LIN {X 0,Y 218.448,Z 342.659,A -85,B 0,C 180,E1 -22368.616,E2 -22368.616} C_VEL
LIN {X 0,Y 217.476,Z 348.635,A -85,B 0,C 180,E1 -22368.653,E2 -22368.653} C_VEL
LIN {X 0,Y 215.786,Z 367.504,A -85,B 0,C 180,E1 -22369.355,E2 -22369.355} C_VEL
LIN {X 0,Y 213.676,Z 380.389,A -85,B 0,C 180,E1 -22370.107,E2 -22370.107} C_VEL
LIN {X 0,Y 210.515,Z 393.733,A -85,B 0,C 180,E1 -22371.248,E2 -22371.248} C_VEL
LIN {X 0,Y 207.06,Z 405.5,A -85,B 0,C 180,E1 -22372.649,E2 -22372.649} C_VEL
LIN {X 0,Y 203.22,Z 416.165,A -85,B 0,C 180,E1 -22374.298,E2 -22374.298} C_VEL
LIN {X 0,Y 199.229,Z 425.901,A -85,B 0,C 180,E1 -22376.249,E2 -22376.249} C_VEL
LIN {X 0,Y 195.179,Z 434.841,A -85,B 0,C 180,E1 -22378.527,E2 -22378.527} C_VEL
LIN {X 0,Y 190.718,Z 443.631,A -85,B 0,C 180,E1 -22381.377,E2 -22381.377} C_VEL
LIN {X 0,Y 186.992,Z 450.647,A -85,B 0,C 180,E1 -22384.353,E2 -22384.353} C_VEL
LIN {X 0,Y 183.667,Z 456.423,A -85,B 0,C 180,E1 -22387.503,E2 -22387.503} C_VEL
LIN {X 0,Y 180.963,Z 460.965,A -85,B 0,C 180,E1 -22390.725,E2 -22390.725} C_VEL
LIN {X 0,Y 178.739,Z 464.46,A -85,B 0,C 180,E1 -22394.024,E2 -22394.024} C_VEL
LIN {X 0,Y 176.979,Z 467.604,A -85,B 0,C 180,E1 -22398.548,E2 -22398.548} C_VEL
LIN {X 0,Y 176.111,Z 469.188,A -85,B 0,C 180,E1 -22403.124,E2 -22403.124} C_VEL
LIN {X 0,Y 175.999,Z 469.294,A -85,B 0,C 180,E1 -22406.825,E2 -22406.825} C_VEL
LIN {X 0,Y 176.229,Z 468.533,A -85,B 0,C 180,E1 -22410,E2 -22410} C_VEL
LIN {X 0,Y 176.089,Z 466.648,A -85,B 0,C 180,E1 -22413.663,E2 -22413.663} C_VEL
LIN {X 0,Y 176.336,Z 462.93,A -85,B 0,C 180,E1 -22418.019,E2 -22418.019} C_VEL
LIN {X 0,Y 176.923,Z 458.748,A -85,B 0,C 180,E1 -22421.456,E2 -22421.456} C_VEL
LIN {X 0,Y 178.216,Z 452.316,A -85,B 0,C 180,E1 -22425.437,E2 -22425.437} C_VEL
LIN {X 0,Y 180.018,Z 445.292,A -85,B 0,C 180,E1 -22428.789,E2 -22428.789} C_VEL
LIN {X 0,Y 181.778,Z 438.618,A -85,B 0,C 180,E1 -22431.344,E2 -22431.344} C_VEL
LIN {X 0,Y 184.193,Z 429.348,A -85,B 0,C 180,E1 -22434.215,E2 -22434.215} C_VEL
LIN {X 0,Y 186.584,Z 419.767,A -85,B 0,C 180,E1 -22436.569,E2 -22436.569} C_VEL
LIN {X 0,Y 188.379,Z 412.204,A -85,B 0,C 180,E1 -22438.099,E2 -22438.099} C_VEL
LIN {X 0,Y 190.939,Z 399.705,A -85,B 0,C 180,E1 -22440.099,E2 -22440.099} C_VEL
LIN {X 0,Y 193.124,Z 387.562,A -85,B 0,C 180,E1 -22441.541,E2 -22441.541} C_VEL
LIN {X 0,Y 194.875,Z 374.064,A -85,B 0,C 180,E1 -22442.672,E2 -22442.672} C_VEL
LIN {X 0,Y 196.016,Z 361.06,A -85,B 0,C 180,E1 -22443.361,E2 -22443.361} C_VEL
LIN {X 0,Y 198.16,Z 316.515,A -85,B 0,C 180,E1 -22445.049,E2 -22445.049} C_VEL
LIN {X 0,Y 195.778,Z 296.397,A -85,B 0,C 180,E1 -22446.33,E2 -22446.33} C_VEL
LIN {X 0,Y 188.073,Z 275.885,A -85,B 0,C 180,E1 -22448.617,E2 -22448.617} C_VEL
LIN {X 0,Y 181.122,Z 260.53,A -85,B 0,C 180,E1 -22450.71,E2 -22450.71} C_VEL
LIN {X 0,Y 179.58,Z 257.045,A -85,B 0,C 180,E1 -22451.221,E2 -22451.221} C_VEL
LIN {X 0,Y 178.411,Z 252.269,A -85,B 0,C 180,E1 -22454.021,E2 -22454.021} C_VEL
LIN {X 0,Y 178.409,Z 252.262,A -85,B 0,C 180,E1 -22458.456,E2 -22458.456} C_VEL
LIN {X 0,Y 178.434,Z 252.257,A -85,B 0,C 180,E1 -22463.773,E2 -22463.773} C_VEL
LIN {X 0,Y 178.497,Z 252.253,A -85,B 0,C 180,E1 -22466.536,E2 -22466.536} C_VEL
LIN {X 0,Y 178.432,Z 252.258,A -85,B 0,C 180,E1 -22471.781,E2 -22471.781} C_VEL
LIN {X 0,Y 178.473,Z 252.253,A -85,B 0,C 180,E1 -22476.797,E2 -22476.797} C_VEL
LIN {X 0,Y 178.613,Z 252.201,A -85,B 0,C 180,E1 -22481.64,E2 -22481.64} C_VEL
LIN {X 0,Y 178.64,Z 252.227,A -85,B 0,C 180,E1 -22486.334,E2 -22486.334} C_VEL
LIN {X 0,Y 178.902,Z 252.196,A -85,B 0,C 180,E1 -22490.947,E2 -22490.947} C_VEL
LIN {X 0,Y 179.098,Z 252.128,A -85,B 0,C 180,E1 -22497.738,E2 -22497.738} C_VEL
LIN {X 0,Y 179.333,Z 252.122,A -85,B 0,C 180,E1 -22499.987,E2 -22499.987} C_VEL
LIN {X 0,Y 178.824,Z 252.209,A -85,B 0,C 180,E1 -22504.495,E2 -22504.495} C_VEL
LIN {X 0,Y 178.893,Z 252.189,A -85,B 0,C 180,E1 -22509.028,E2 -22509.028} C_VEL
LIN {X 0,Y 178.636,Z 252.234,A -85,B 0,C 180,E1 -22513.64,E2 -22513.64} C_VEL
LIN {X 0,Y 178.603,Z 252.223,A -85,B 0,C 180,E1 -22519.2,E2 -22519.2} C_VEL
LIN {X 0,Y 178.497,Z 252.245,A -85,B 0,C 180,E1 -22525.101,E2 -22525.101} C_VEL
LIN {X 0,Y 178.437,Z 252.208,A -85,B 0,C 180,E1 -22530.782,E2 -22530.782} C_VEL
LIN {X 0,Y 178.453,Z 252.224,A -85,B 0,C 180,E1 -22534.206,E2 -22534.206} C_VEL
LIN {X 0,Y 178.356,Z 252.267,A -85,B 0,C 180,E1 -22539.065,E2 -22539.065} C_VEL
LIN {X 0,Y 178.361,Z 252.261,A -85,B 0,C 180,E1 -22542.036,E2 -22542.036} C_VEL
LIN {X 0,Y 178.357,Z 252.263,A -85,B 0,C 180,E1 -22545.154,E2 -22545.154} C_VEL
LIN {X 0,Y 178.365,Z 252.265,A -85,B 0,C 180,E1 -22548.45,E2 -22548.45} C_VEL
LIN {X 0,Y 178.381,Z 252.266,A -85,B 0,C 180,E1 -22553.774,E2 -22553.774} C_VEL
LIN {X 0,Y 178.443,Z 252.252,A -85,B 0,C 180,E1 -22556.538,E2 -22556.538} C_VEL
LIN {X 0,Y 178.479,Z 252.256,A -85,B 0,C 180,E1 -22560,E2 -22560} C_VEL
LIN {X 0,Y 178.5,Z 252.256,A -85,B 0,C 180,E1 -22564.863,E2 -22564.863} C_VEL
LIN {X 0,Y 178.608,Z 252.243,A -85,B 0,C 180,E1 -22570.75,E2 -22570.75} C_VEL
LIN {X 0,Y 178.626,Z 252.239,A -85,B 0,C 180,E1 -22574.014,E2 -22574.014} C_VEL
LIN {X 0,Y 178.81,Z 252.209,A -85,B 0,C 180,E1 -22579.213,E2 -22579.213} C_VEL
LIN {X 0,Y 178.907,Z 252.197,A -85,B 0,C 180,E1 -22582.026,E2 -22582.026} C_VEL
LIN {X 0,Y 179.914,Z 255.085,A -85,B 0,C 180,E1 -22582.417,E2 -22582.417} C_VEL
LIN {X 0,Y 181.316,Z 257.484,A -85,B 0,C 180,E1 -22582.826,E2 -22582.826} C_VEL
LIN {X 0,Y 189.994,Z 273.152,A -85,B 0,C 180,E1 -22585.256,E2 -22585.256} C_VEL
LIN {X 0,Y 194.262,Z 282.713,A -85,B 0,C 180,E1 -22586.448,E2 -22586.448} C_VEL
LIN {X 0,Y 199.123,Z 295.475,A -85,B 0,C 180,E1 -22587.811,E2 -22587.811} C_VEL
LIN {X 0,Y 195.994,Z 353.238,A -85,B 0,C 180,E1 -22590,E2 -22590} C_VEL
LIN {X 0,Y 194.697,Z 366.02,A -85,B 0,C 180,E1 -22590.84,E2 -22590.84} C_VEL
LIN {X 0,Y 193.136,Z 378.634,A -85,B 0,C 180,E1 -22592.085,E2 -22592.085} C_VEL
LIN {X 0,Y 191.05,Z 390.66,A -85,B 0,C 180,E1 -22593.691,E2 -22593.691} C_VEL
LIN {X 0,Y 188.528,Z 402.811,A -85,B 0,C 180,E1 -22595.83,E2 -22595.83} C_VEL
LIN {X 0,Y 186.128,Z 413.03,A -85,B 0,C 180,E1 -22598.14,E2 -22598.14} C_VEL
LIN {X 0,Y 183.418,Z 423.131,A -85,B 0,C 180,E1 -22601.045,E2 -22601.045} C_VEL
LIN {X 0,Y 181.186,Z 431.752,A -85,B 0,C 180,E1 -22604.201,E2 -22604.201} C_VEL
LIN {X 0,Y 179.205,Z 439.195,A -85,B 0,C 180,E1 -22607.694,E2 -22607.694} C_VEL
LIN {X 0,Y 177.904,Z 444.467,A -85,B 0,C 180,E1 -22610.826,E2 -22610.826} C_VEL
LIN {X 0,Y 176.83,Z 449.719,A -85,B 0,C 180,E1 -22614.916,E2 -22614.916} C_VEL
LIN {X 0,Y 176.035,Z 453.133,A -85,B 0,C 180,E1 -22618.625,E2 -22618.625} C_VEL
LIN {X 0,Y 175.672,Z 455.615,A -85,B 0,C 180,E1 -22622.875,E2 -22622.875} C_VEL
LIN {X 0,Y 175.993,Z 456.678,A -85,B 0,C 180,E1 -22627.023,E2 -22627.023} C_VEL
LIN {X 0,Y 176.857,Z 456.49,A -85,B 0,C 180,E1 -22630.996,E2 -22630.996} C_VEL
LIN {X 0,Y 178.438,Z 455.004,A -85,B 0,C 180,E1 -22635.148,E2 -22635.148} C_VEL
LIN {X 0,Y 180.843,Z 451.875,A -85,B 0,C 180,E1 -22639.502,E2 -22639.502} C_VEL
LIN {X 0,Y 183.816,Z 447.528,A -85,B 0,C 180,E1 -22643.407,E2 -22643.407} C_VEL
LIN {X 0,Y 187.038,Z 442.414,A -85,B 0,C 180,E1 -22646.722,E2 -22646.722} C_VEL
LIN {X 0,Y 190.908,Z 435.903,A -85,B 0,C 180,E1 -22649.891,E2 -22649.891} C_VEL
LIN {X 0,Y 194.765,Z 428.674,A -85,B 0,C 180,E1 -22652.617,E2 -22652.617} C_VEL
LIN {X 0,Y 199.095,Z 419.632,A -85,B 0,C 180,E1 -22655.279,E2 -22655.279} C_VEL
LIN {X 0,Y 203.103,Z 410.186,A -85,B 0,C 180,E1 -22657.463,E2 -22657.463} C_VEL
LIN {X 0,Y 206.676,Z 400.411,A -85,B 0,C 180,E1 -22659.246,E2 -22659.246} C_VEL
LIN {X 0,Y 210.237,Z 388.81,A -85,B 0,C 180,E1 -22660.877,E2 -22660.877} C_VEL
LIN {X 0,Y 213.117,Z 377.076,A -85,B 0,C 180,E1 -22662.134,E2 -22662.134} C_VEL
LIN {X 0,Y 215.495,Z 364.012,A -85,B 0,C 180,E1 -22663.149,E2 -22663.149} C_VEL
LIN {X 0,Y 217.106,Z 350.758,A -85,B 0,C 180,E1 -22663.799,E2 -22663.799} C_VEL
LIN {X 0,Y 220.108,Z 311.417,A -85,B 0,C 180,E1 -22665.133,E2 -22665.133} C_VEL
LIN {X 0,Y 216.218,Z 302.782,A -85,B 0,C 180,E1 -22667.007,E2 -22667.007} C_VEL
LIN {X 0,Y 213.125,Z 297.063,A -85,B 0,C 180,E1 -22668.556,E2 -22668.556} C_VEL
LIN {X 0,Y 209.272,Z 290.775,A -85,B 0,C 180,E1 -22670.62,E2 -22670.62} C_VEL
LIN {X 0,Y 204.339,Z 283.304,A -85,B 0,C 180,E1 -22673.596,E2 -22673.596} C_VEL
LIN {X 0,Y 201.792,Z 279.641,A -85,B 0,C 180,E1 -22675.355,E2 -22675.355} C_VEL
LIN {X 0,Y 199.009,Z 276.05,A -85,B 0,C 180,E1 -22677.458,E2 -22677.458} C_VEL
LIN {X 0,Y 198.122,Z 274.662,A -85,B 0,C 180,E1 -22678.233,E2 -22678.233} C_VEL
LIN {X 0,Y 195.806,Z 271.796,A -85,B 0,C 180,E1 -22680.344,E2 -22680.344} C_VEL
LIN {X 0,Y 194.667,Z 269.788,A -85,B 0,C 180,E1 -22681.573,E2 -22681.573} C_VEL
LIN {X 0,Y 191.537,Z 267.402,A -85,B 0,C 180,E1 -22685.275,E2 -22685.275} C_VEL
LIN {X 0,Y 190.259,Z 264.56,A -85,B 0,C 180,E1 -22687.635,E2 -22687.635} C_VEL
LIN {X 0,Y 188.459,Z 263.748,A -85,B 0,C 180,E1 -22691.847,E2 -22691.847} C_VEL
LIN {X 0,Y 187.853,Z 263.472,A -85,B 0,C 180,E1 -22697.427,E2 -22697.427} C_VEL
LIN {X 0,Y 189.234,Z 264.37,A -85,B 0,C 180,E1 -22702.926,E2 -22702.926} C_VEL
LIN {X 0,Y 190.557,Z 266.295,A -85,B 0,C 180,E1 -22705.656,E2 -22705.656} C_VEL
LIN {X 0,Y 192.69,Z 269.516,A -85,B 0,C 180,E1 -22708.916,E2 -22708.916} C_VEL
LIN {X 0,Y 195.62,Z 273.297,A -85,B 0,C 180,E1 -22712.167,E2 -22712.167} C_VEL
LIN {X 0,Y 199.882,Z 279.881,A -85,B 0,C 180,E1 -22715.981,E2 -22715.981} C_VEL
LIN {X 0,Y 203.656,Z 286.092,A -85,B 0,C 180,E1 -22718.753,E2 -22718.753} C_VEL
LIN {X 0,Y 206.674,Z 291.312,A -85,B 0,C 180,E1 -22720.699,E2 -22720.699} C_VEL
LIN {X 0,Y 210.875,Z 299.125,A -85,B 0,C 180,E1 -22723.158,E2 -22723.158} C_VEL
LIN {X 0,Y 215.414,Z 308.937,A -85,B 0,C 180,E1 -22725.57,E2 -22725.57} C_VEL
LIN {X 0,Y 219.144,Z 318.713,A -85,B 0,C 180,E1 -22727.455,E2 -22727.455} C_VEL
LIN {X 0,Y 219.436,Z 321.912,A -85,B 0,C 180,E1 -22727.735,E2 -22727.735} C_VEL
LIN {X 0,Y 217.476,Z 348.635,A -85,B 0,C 180,E1 -22728.653,E2 -22728.653} C_VEL
LIN {X 0,Y 216.967,Z 352.543,A -85,B 0,C 180,E1 -22728.712,E2 -22728.712} C_VEL
LIN {X 0,Y 214.974,Z 360.206,A -85,B 0,C 180,E1 -22728.535,E2 -22728.535} C_VEL
LIN {X 0,Y 211.006,Z 371.945,A -85,B 0,C 180,E1 -22728.28,E2 -22728.28} C_VEL
LIN {X 0,Y 209.635,Z 377.18,A -85,B 0,C 180,E1 -22728.446,E2 -22728.446} C_VEL
LIN {X 0,Y 209.282,Z 379.016,A -85,B 0,C 180,E1 -22728.568,E2 -22728.568} C_VEL
LIN {X 0,Y 206.137,Z 392.042,A -85,B 0,C 180,E1 -22729.627,E2 -22729.627} C_VEL
LIN {X 0,Y 202.56,Z 404.078,A -85,B 0,C 180,E1 -22731.035,E2 -22731.035} C_VEL
LIN {X 0,Y 198.538,Z 414.999,A -85,B 0,C 180,E1 -22732.686,E2 -22732.686} C_VEL
LIN {X 0,Y 194.324,Z 424.911,A -85,B 0,C 180,E1 -22734.645,E2 -22734.645} C_VEL
LIN {X 0,Y 189.996,Z 433.938,A -85,B 0,C 180,E1 -22736.935,E2 -22736.935} C_VEL
LIN {X 0,Y 185.284,Z 442.796,A -85,B 0,C 180,E1 -22739.83,E2 -22739.83} C_VEL
LIN {X 0,Y 181.174,Z 449.989,A -85,B 0,C 180,E1 -22742.885,E2 -22742.885} C_VEL
LIN {X 0,Y 178.262,Z 454.888,A -85,B 0,C 180,E1 -22745.547,E2 -22745.547} C_VEL
LIN {X 0,Y 175.186,Z 459.697,A -85,B 0,C 180,E1 -22748.836,E2 -22748.836} C_VEL
LIN {X 0,Y 172.634,Z 463.423,A -85,B 0,C 180,E1 -22752.223,E2 -22752.223} C_VEL
LIN {X 0,Y 170.812,Z 466.166,A -85,B 0,C 180,E1 -22755.708,E2 -22755.708} C_VEL
LIN {X 0,Y 169.394,Z 468.429,A -85,B 0,C 180,E1 -22760.448,E2 -22760.448} C_VEL
LIN {X 0,Y 168.954,Z 469.072,A -85,B 0,C 180,E1 -22765.228,E2 -22765.228} C_VEL
LIN {X 0,Y 168.957,Z 468.811,A -85,B 0,C 180,E1 -22767.616,E2 -22767.616} C_VEL
LIN {X 0,Y 169.131,Z 468.163,A -85,B 0,C 180,E1 -22770,E2 -22770} C_VEL
LIN {X 0,Y 169.004,Z 466.426,A -85,B 0,C 180,E1 -22773.428,E2 -22773.428} C_VEL
LIN {X 0,Y 169.292,Z 462.334,A -85,B 0,C 180,E1 -22778.355,E2 -22778.355} C_VEL
LIN {X 0,Y 169.941,Z 458.05,A -85,B 0,C 180,E1 -22781.933,E2 -22781.933} C_VEL
LIN {X 0,Y 171.35,Z 451.51,A -85,B 0,C 180,E1 -22786.072,E2 -22786.072} C_VEL
LIN {X 0,Y 173.261,Z 444.307,A -85,B 0,C 180,E1 -22789.551,E2 -22789.551} C_VEL
LIN {X 0,Y 174.884,Z 438.404,A -85,B 0,C 180,E1 -22791.878,E2 -22791.878} C_VEL
LIN {X 0,Y 177.204,Z 430,A -85,B 0,C 180,E1 -22794.609,E2 -22794.609} C_VEL
LIN {X 0,Y 179.627,Z 420.604,A -85,B 0,C 180,E1 -22797.054,E2 -22797.054} C_VEL
LIN {X 0,Y 181.399,Z 413.157,A -85,B 0,C 180,E1 -22798.649,E2 -22798.649} C_VEL
LIN {X 0,Y 183.744,Z 402.8,A -85,B 0,C 180,E1 -22800.45,E2 -22800.45} C_VEL
LIN {X 0,Y 186.156,Z 390.494,A -85,B 0,C 180,E1 -22802.066,E2 -22802.066} C_VEL
LIN {X 0,Y 188.093,Z 376.919,A -85,B 0,C 180,E1 -22803.363,E2 -22803.363} C_VEL
LIN {X 0,Y 189.452,Z 364.232,A -85,B 0,C 180,E1 -22804.136,E2 -22804.136} C_VEL
LIN {X 0,Y 191.835,Z 317.292,A -85,B 0,C 180,E1 -22805.99,E2 -22805.99} C_VEL
LIN {X 0,Y 189.723,Z 298.628,A -85,B 0,C 180,E1 -22807.221,E2 -22807.221} C_VEL
LIN {X 0,Y 182.321,Z 278.848,A -85,B 0,C 180,E1 -22809.545,E2 -22809.545} C_VEL
LIN {X 0,Y 175.933,Z 264.533,A -85,B 0,C 180,E1 -22811.576,E2 -22811.576} C_VEL
LIN {X 0,Y 172.205,Z 256.731,A -85,B 0,C 180,E1 -22812.835,E2 -22812.835} C_VEL
LIN {X 0,Y 171.373,Z 253.141,A -85,B 0,C 180,E1 -22815.108,E2 -22815.108} C_VEL
LIN {X 0,Y 171.343,Z 253.142,A -85,B 0,C 180,E1 -22818.969,E2 -22818.969} C_VEL
LIN {X 0,Y 171.376,Z 253.14,A -85,B 0,C 180,E1 -22822.024,E2 -22822.024} C_VEL
LIN {X 0,Y 171.413,Z 253.134,A -85,B 0,C 180,E1 -22825.083,E2 -22825.083} C_VEL
LIN {X 0,Y 171.402,Z 253.136,A -85,B 0,C 180,E1 -22830.512,E2 -22830.512} C_VEL
LIN {X 0,Y 171.413,Z 253.134,A -85,B 0,C 180,E1 -22835.782,E2 -22835.782} C_VEL
LIN {X 0,Y 171.516,Z 253.088,A -85,B 0,C 180,E1 -22840.851,E2 -22840.851} C_VEL
LIN {X 0,Y 171.555,Z 253.104,A -85,B 0,C 180,E1 -22845.758,E2 -22845.758} C_VEL
LIN {X 0,Y 171.842,Z 253.076,A -85,B 0,C 180,E1 -22850.572,E2 -22850.572} C_VEL
LIN {X 0,Y 171.758,Z 253.042,A -85,B 0,C 180,E1 -22855.293,E2 -22855.293} C_VEL
LIN {X 0,Y 172.298,Z 252.997,A -85,B 0,C 180,E1 -22859.987,E2 -22859.987} C_VEL
LIN {X 0,Y 171.774,Z 253.087,A -85,B 0,C 180,E1 -22864.68,E2 -22864.68} C_VEL
LIN {X 0,Y 171.831,Z 253.067,A -85,B 0,C 180,E1 -22869.402,E2 -22869.402} C_VEL
LIN {X 0,Y 171.553,Z 253.114,A -85,B 0,C 180,E1 -22874.215,E2 -22874.215} C_VEL
LIN {X 0,Y 171.521,Z 253.106,A -85,B 0,C 180,E1 -22879.543,E2 -22879.543} C_VEL
LIN {X 0,Y 171.434,Z 253.121,A -85,B 0,C 180,E1 -22885.594,E2 -22885.594} C_VEL
LIN {X 0,Y 171.394,Z 253.084,A -85,B 0,C 180,E1 -22890.562,E2 -22890.562} C_VEL
LIN {X 0,Y 171.363,Z 253.116,A -85,B 0,C 180,E1 -22895.023,E2 -22895.023} C_VEL
LIN {X 0,Y 171.312,Z 253.144,A -85,B 0,C 180,E1 -22898.79,E2 -22898.79} C_VEL
LIN {X 0,Y 171.284,Z 253.141,A -85,B 0,C 180,E1 -22904.207,E2 -22904.207} C_VEL
LIN {X 0,Y 171.297,Z 253.143,A -85,B 0,C 180,E1 -22908.971,E2 -22908.971} C_VEL
LIN {X 0,Y 171.346,Z 253.14,A -85,B 0,C 180,E1 -22912.031,E2 -22912.031} C_VEL
LIN {X 0,Y 171.357,Z 253.139,A -85,B 0,C 180,E1 -22915.084,E2 -22915.084} C_VEL
LIN {X 0,Y 171.406,Z 253.138,A -85,B 0,C 180,E1 -22920.527,E2 -22920.527} C_VEL
LIN {X 0,Y 171.427,Z 253.136,A -85,B 0,C 180,E1 -22925.798,E2 -22925.798} C_VEL
LIN {X 0,Y 171.564,Z 253.119,A -85,B 0,C 180,E1 -22930.87,E2 -22930.87} C_VEL
LIN {X 0,Y 171.548,Z 253.114,A -85,B 0,C 180,E1 -22935.771,E2 -22935.771} C_VEL
LIN {X 0,Y 171.821,Z 253.081,A -85,B 0,C 180,E1 -22940.518,E2 -22940.518} C_VEL
LIN {X 0,Y 172.984,Z 256.112,A -85,B 0,C 180,E1 -22940.99,E2 -22940.99} C_VEL
LIN {X 0,Y 174.215,Z 258.076,A -85,B 0,C 180,E1 -22941.369,E2 -22941.369} C_VEL
LIN {X 0,Y 185.194,Z 278.048,A -85,B 0,C 180,E1 -22944.616,E2 -22944.616} C_VEL
LIN {X 0,Y 189.645,Z 288.755,A -85,B 0,C 180,E1 -22945.947,E2 -22945.947} C_VEL
LIN {X 0,Y 192.884,Z 297.515,A -85,B 0,C 180,E1 -22946.911,E2 -22946.911} C_VEL
LIN {X 0,Y 189.603,Z 353.724,A -85,B 0,C 180,E1 -22949.09,E2 -22949.09} C_VEL
LIN {X 0,Y 188.26,Z 366.475,A -85,B 0,C 180,E1 -22949.957,E2 -22949.957} C_VEL
LIN {X 0,Y 186.662,Z 378.826,A -85,B 0,C 180,E1 -22951.213,E2 -22951.213} C_VEL
LIN {X 0,Y 184.693,Z 389.908,A -85,B 0,C 180,E1 -22952.711,E2 -22952.711} C_VEL
LIN {X 0,Y 182.311,Z 401.179,A -85,B 0,C 180,E1 -22954.699,E2 -22954.699} C_VEL
LIN {X 0,Y 179.832,Z 411.506,A -85,B 0,C 180,E1 -22957.015,E2 -22957.015} C_VEL
LIN {X 0,Y 177.211,Z 421.08,A -85,B 0,C 180,E1 -22959.703,E2 -22959.703} C_VEL
LIN {X 0,Y 174.899,Z 429.64,A -85,B 0,C 180,E1 -22962.768,E2 -22962.768} C_VEL
LIN {X 0,Y 172.61,Z 437.952,A -85,B 0,C 180,E1 -22966.559,E2 -22966.559} C_VEL
LIN {X 0,Y 170.893,Z 444.529,A -85,B 0,C 180,E1 -22970.485,E2 -22970.485} C_VEL
LIN {X 0,Y 169.81,Z 449.528,A -85,B 0,C 180,E1 -22974.462,E2 -22974.462} C_VEL
LIN {X 0,Y 169.182,Z 452.182,A -85,B 0,C 180,E1 -22977.19,E2 -22977.19} C_VEL
LIN {X 0,Y 168.726,Z 454.227,A -85,B 0,C 180,E1 -22979.988,E2 -22979.988} C_VEL
LIN {X 0,Y 168.607,Z 456.019,A -85,B 0,C 180,E1 -22983.553,E2 -22983.553} C_VEL
LIN {X 0,Y 169.01,Z 456.981,A -85,B 0,C 180,E1 -22987.833,E2 -22987.833} C_VEL
LIN {X 0,Y 170.012,Z 456.715,A -85,B 0,C 180,E1 -22991.943,E2 -22991.943} C_VEL
LIN {X 0,Y 171.624,Z 455.317,A -85,B 0,C 180,E1 -22995.903,E2 -22995.903} C_VEL
LIN {X 0,Y 174.032,Z 452.498,A -85,B 0,C 180,E1 -23000.109,E2 -23000.109} C_VEL
LIN {X 0,Y 177.436,Z 447.916,A -85,B 0,C 180,E1 -23004.426,E2 -23004.426} C_VEL
LIN {X 0,Y 180.504,Z 443.361,A -85,B 0,C 180,E1 -23007.52,E2 -23007.52} C_VEL
LIN {X 0,Y 184.821,Z 436.597,A -85,B 0,C 180,E1 -23010.994,E2 -23010.994} C_VEL
LIN {X 0,Y 189.414,Z 428.473,A -85,B 0,C 180,E1 -23014.124,E2 -23014.124} C_VEL
LIN {X 0,Y 193.781,Z 419.832,A -85,B 0,C 180,E1 -23016.696,E2 -23016.696} C_VEL
LIN {X 0,Y 198.269,Z 409.678,A -85,B 0,C 180,E1 -23019.047,E2 -23019.047} C_VEL
LIN {X 0,Y 202.389,Z 398.642,A -85,B 0,C 180,E1 -23021,E2 -23021} C_VEL
LIN {X 0,Y 205.619,Z 388.374,A -85,B 0,C 180,E1 -23022.41,E2 -23022.41} C_VEL
LIN {X 0,Y 208.694,Z 376.223,A -85,B 0,C 180,E1 -23023.687,E2 -23023.687} C_VEL
LIN {X 0,Y 211.121,Z 362.816,A -85,B 0,C 180,E1 -23024.693,E2 -23024.693} C_VEL
LIN {X 0,Y 212.823,Z 348.84,A -85,B 0,C 180,E1 -23025.335,E2 -23025.335} C_VEL
LIN {X 0,Y 215.641,Z 314.414,A -85,B 0,C 180,E1 -23026.481,E2 -23026.481} C_VEL
LIN {X 0,Y 211.748,Z 305.602,A -85,B 0,C 180,E1 -23028.525,E2 -23028.525} C_VEL
LIN {X 0,Y 206.997,Z 297.301,A -85,B 0,C 180,E1 -23031.169,E2 -23031.169} C_VEL
LIN {X 0,Y 201.996,Z 289.45,A -85,B 0,C 180,E1 -23034.349,E2 -23034.349} C_VEL
LIN {X 0,Y 199.601,Z 285.928,A -85,B 0,C 180,E1 -23036.092,E2 -23036.092} C_VEL
LIN {X 0,Y 196.898,Z 282.215,A -85,B 0,C 180,E1 -23038.28,E2 -23038.28} C_VEL
LIN {X 0,Y 195.875,Z 280.804,A -85,B 0,C 180,E1 -23039.208,E2 -23039.208} C_VEL
LIN {X 0,Y 193.625,Z 277.529,A -85,B 0,C 180,E1 -23041.474,E2 -23041.474} C_VEL
LIN {X 0,Y 193.079,Z 276.565,A -85,B 0,C 180,E1 -23042.098,E2 -23042.098} C_VEL
LIN {X 0,Y 190.114,Z 274.095,A -85,B 0,C 180,E1 -23045.846,E2 -23045.846} C_VEL
LIN {X 0,Y 188.953,Z 271.398,A -85,B 0,C 180,E1 -23048.168,E2 -23048.168} C_VEL
LIN {X 0,Y 186.835,Z 270.456,A -85,B 0,C 180,E1 -23055.278,E2 -23055.278} C_VEL
LIN {X 0,Y 187.857,Z 271.064,A -85,B 0,C 180,E1 -23061.981,E2 -23061.981} C_VEL
LIN {X 0,Y 189.203,Z 273.014,A -85,B 0,C 180,E1 -23065.098,E2 -23065.098} C_VEL
LIN {X 0,Y 191.427,Z 276.579,A -85,B 0,C 180,E1 -23068.665,E2 -23068.665} C_VEL
LIN {X 0,Y 193.817,Z 279.733,A -85,B 0,C 180,E1 -23071.458,E2 -23071.458} C_VEL
LIN {X 0,Y 197.728,Z 286.127,A -85,B 0,C 180,E1 -23075.206,E2 -23075.206} C_VEL
LIN {X 0,Y 201.329,Z 292.293,A -85,B 0,C 180,E1 -23078.013,E2 -23078.013} C_VEL
LIN {X 0,Y 203.915,Z 297.017,A -85,B 0,C 180,E1 -23079.796,E2 -23079.796} C_VEL
LIN {X 0,Y 207.947,Z 304.892,A -85,B 0,C 180,E1 -23082.315,E2 -23082.315} C_VEL
LIN {X 0,Y 211.961,Z 313.976,A -85,B 0,C 180,E1 -23084.594,E2 -23084.594} C_VEL
LIN {X 0,Y 214.928,Z 322.373,A -85,B 0,C 180,E1 -23086.242,E2 -23086.242} C_VEL
LIN {X 0,Y 213.906,Z 337.035,A -85,B 0,C 180,E1 -23086.794,E2 -23086.794} C_VEL
LIN {X 0,Y 211.489,Z 365.432,A -85,B 0,C 180,E1 -23087.808,E2 -23087.808} C_VEL
LIN {X 0,Y 209.282,Z 379.016,A -85,B 0,C 180,E1 -23088.568,E2 -23088.568} C_VEL
LIN {X 0,Y 207.785,Z 384.62,A -85,B 0,C 180,E1 -23088.868,E2 -23088.868} C_VEL
LIN {X 0,Y 203.597,Z 393.586,A -85,B 0,C 180,E1 -23089.074,E2 -23089.074} C_VEL
LIN {X 0,Y 198.88,Z 402.223,A -85,B 0,C 180,E1 -23089.43,E2 -23089.43} C_VEL
LIN {X 0,Y 196.574,Z 407.309,A -85,B 0,C 180,E1 -23089.981,E2 -23089.981} C_VEL
LIN {X 0,Y 192.002,Z 418.533,A -85,B 0,C 180,E1 -23091.854,E2 -23091.854} C_VEL
LIN {X 0,Y 187.685,Z 427.792,A -85,B 0,C 180,E1 -23093.861,E2 -23093.861} C_VEL
LIN {X 0,Y 183.308,Z 436.293,A -85,B 0,C 180,E1 -23096.227,E2 -23096.227} C_VEL
LIN {X 0,Y 178.454,Z 444.623,A -85,B 0,C 180,E1 -23099.206,E2 -23099.206} C_VEL
LIN {X 0,Y 174.13,Z 451.581,A -85,B 0,C 180,E1 -23102.476,E2 -23102.476} C_VEL
LIN {X 0,Y 170.642,Z 456.829,A -85,B 0,C 180,E1 -23105.679,E2 -23105.679} C_VEL
LIN {X 0,Y 167.618,Z 461.146,A -85,B 0,C 180,E1 -23109.122,E2 -23109.122} C_VEL
LIN {X 0,Y 165.1,Z 464.442,A -85,B 0,C 180,E1 -23112.665,E2 -23112.665} C_VEL
LIN {X 0,Y 163.023,Z 467.388,A -85,B 0,C 180,E1 -23117.553,E2 -23117.553} C_VEL
LIN {X 0,Y 162.383,Z 468.245,A -85,B 0,C 180,E1 -23120.031,E2 -23120.031} C_VEL
LIN {X 0,Y 161.871,Z 468.784,A -85,B 0,C 180,E1 -23125.019,E2 -23125.019} C_VEL
LIN {X 0,Y 161.867,Z 468.481,A -85,B 0,C 180,E1 -23127.512,E2 -23127.512} C_VEL
LIN {X 0,Y 162.035,Z 467.776,A -85,B 0,C 180,E1 -23130,E2 -23130} C_VEL
LIN {X 0,Y 161.909,Z 466.252,A -85,B 0,C 180,E1 -23133.087,E2 -23133.087} C_VEL
LIN {X 0,Y 162.098,Z 462.965,A -85,B 0,C 180,E1 -23137.474,E2 -23137.474} C_VEL
LIN {X 0,Y 162.664,Z 458.967,A -85,B 0,C 180,E1 -23141.211,E2 -23141.211} C_VEL
LIN {X 0,Y 163.957,Z 452.751,A -85,B 0,C 180,E1 -23145.539,E2 -23145.539} C_VEL
LIN {X 0,Y 165.836,Z 445.947,A -85,B 0,C 180,E1 -23149.174,E2 -23149.174} C_VEL
LIN {X 0,Y 167.815,Z 438.987,A -85,B 0,C 180,E1 -23152.142,E2 -23152.142} C_VEL
LIN {X 0,Y 169.687,Z 432.393,A -85,B 0,C 180,E1 -23154.467,E2 -23154.467} C_VEL
LIN {X 0,Y 172.419,Z 422.504,A -85,B 0,C 180,E1 -23157.294,E2 -23157.294} C_VEL
LIN {X 0,Y 174.823,Z 412.8,A -85,B 0,C 180,E1 -23159.502,E2 -23159.502} C_VEL
LIN {X 0,Y 177.26,Z 402.42,A -85,B 0,C 180,E1 -23161.357,E2 -23161.357} C_VEL
LIN {X 0,Y 179.744,Z 390.062,A -85,B 0,C 180,E1 -23163.021,E2 -23163.021} C_VEL
LIN {X 0,Y 181.771,Z 376.445,A -85,B 0,C 180,E1 -23164.35,E2 -23164.35} C_VEL
LIN {X 0,Y 183.145,Z 363.661,A -85,B 0,C 180,E1 -23165.141,E2 -23165.141} C_VEL
LIN {X 0,Y 185.608,Z 318.285,A -85,B 0,C 180,E1 -23166.975,E2 -23166.975} C_VEL
LIN {X 0,Y 183.654,Z 300.792,A -85,B 0,C 180,E1 -23168.187,E2 -23168.187} C_VEL
LIN {X 0,Y 176.413,Z 281.384,A -85,B 0,C 180,E1 -23170.571,E2 -23170.571} C_VEL
LIN {X 0,Y 170.341,Z 267.741,A -85,B 0,C 180,E1 -23172.622,E2 -23172.622} C_VEL
LIN {X 0,Y 164.846,Z 256.315,A -85,B 0,C 180,E1 -23174.632,E2 -23174.632} C_VEL
LIN {X 0,Y 164.29,Z 254.025,A -85,B 0,C 180,E1 -23176.181,E2 -23176.181} C_VEL
LIN {X 0,Y 164.305,Z 254.019,A -85,B 0,C 180,E1 -23180.346,E2 -23180.346} C_VEL
LIN {X 0,Y 164.342,Z 254.012,A -85,B 0,C 180,E1 -23184.342,E2 -23184.342} C_VEL
LIN {X 0,Y 164.368,Z 254.008,A -85,B 0,C 180,E1 -23189.116,E2 -23189.116} C_VEL
LIN {X 0,Y 164.367,Z 254.008,A -85,B 0,C 180,E1 -23194.672,E2 -23194.672} C_VEL
LIN {X 0,Y 164.425,Z 253.978,A -85,B 0,C 180,E1 -23200.106,E2 -23200.106} C_VEL
LIN {X 0,Y 164.484,Z 253.98,A -85,B 0,C 180,E1 -23205.132,E2 -23205.132} C_VEL
LIN {X 0,Y 164.764,Z 253.958,A -85,B 0,C 180,E1 -23210.163,E2 -23210.163} C_VEL
LIN {X 0,Y 164.814,Z 253.936,A -85,B 0,C 180,E1 -23212.637,E2 -23212.637} C_VEL
LIN {X 0,Y 165.26,Z 253.872,A -85,B 0,C 180,E1 -23219.986,E2 -23219.986} C_VEL
LIN {X 0,Y 164.809,Z 253.949,A -85,B 0,C 180,E1 -23227.336,E2 -23227.336} C_VEL
LIN {X 0,Y 164.69,Z 253.96,A -85,B 0,C 180,E1 -23231.044,E2 -23231.044} C_VEL
LIN {X 0,Y 164.461,Z 253.986,A -85,B 0,C 180,E1 -23237.39,E2 -23237.39} C_VEL
LIN {X 0,Y 164.455,Z 253.989,A -85,B 0,C 180,E1 -23239.975,E2 -23239.975} C_VEL
LIN {X 0,Y 164.359,Z 254,A -85,B 0,C 180,E1 -23246.112,E2 -23246.112} C_VEL
LIN {X 0,Y 164.328,Z 253.959,A -85,B 0,C 180,E1 -23251.203,E2 -23251.203} C_VEL
LIN {X 0,Y 164.249,Z 254.015,A -85,B 0,C 180,E1 -23256.781,E2 -23256.781} C_VEL
LIN {X 0,Y 164.254,Z 254.024,A -85,B 0,C 180,E1 -23259.906,E2 -23259.906} C_VEL
LIN {X 0,Y 164.246,Z 254.015,A -85,B 0,C 180,E1 -23263.331,E2 -23263.331} C_VEL
LIN {X 0,Y 164.226,Z 254.028,A -85,B 0,C 180,E1 -23266.788,E2 -23266.788} C_VEL
LIN {X 0,Y 164.256,Z 254.014,A -85,B 0,C 180,E1 -23270.343,E2 -23270.343} C_VEL
LIN {X 0,Y 164.289,Z 254.021,A -85,B 0,C 180,E1 -23274.34,E2 -23274.34} C_VEL
LIN {X 0,Y 164.346,Z 254.017,A -85,B 0,C 180,E1 -23279.126,E2 -23279.126} C_VEL
LIN {X 0,Y 164.38,Z 254.015,A -85,B 0,C 180,E1 -23284.689,E2 -23284.689} C_VEL
LIN {X 0,Y 164.475,Z 254.004,A -85,B 0,C 180,E1 -23290.011,E2 -23290.011} C_VEL
LIN {X 0,Y 164.5,Z 253.995,A -85,B 0,C 180,E1 -23295.147,E2 -23295.147} C_VEL
LIN {X 0,Y 164.677,Z 253.971,A -85,B 0,C 180,E1 -23298.897,E2 -23298.897} C_VEL
LIN {X 0,Y 165.746,Z 256.867,A -85,B 0,C 180,E1 -23299.341,E2 -23299.341} C_VEL
LIN {X 0,Y 167.259,Z 258.975,A -85,B 0,C 180,E1 -23299.827,E2 -23299.827} C_VEL
LIN {X 0,Y 178.715,Z 279.696,A -85,B 0,C 180,E1 -23303.466,E2 -23303.466} C_VEL
LIN {X 0,Y 182.951,Z 289.23,A -85,B 0,C 180,E1 -23304.761,E2 -23304.761} C_VEL
LIN {X 0,Y 186.623,Z 298.942,A -85,B 0,C 180,E1 -23305.911,E2 -23305.911} C_VEL
LIN {X 0,Y 183.29,Z 353.799,A -85,B 0,C 180,E1 -23308.092,E2 -23308.092} C_VEL
LIN {X 0,Y 181.911,Z 366.503,A -85,B 0,C 180,E1 -23308.973,E2 -23308.973} C_VEL
LIN {X 0,Y 180.224,Z 379.03,A -85,B 0,C 180,E1 -23310.279,E2 -23310.279} C_VEL
LIN {X 0,Y 178.009,Z 391.061,A -85,B 0,C 180,E1 -23311.98,E2 -23311.98} C_VEL
LIN {X 0,Y 175.519,Z 402.149,A -85,B 0,C 180,E1 -23314.024,E2 -23314.024} C_VEL
LIN {X 0,Y 172.986,Z 412.322,A -85,B 0,C 180,E1 -23316.414,E2 -23316.414} C_VEL
LIN {X 0,Y 170.404,Z 421.343,A -85,B 0,C 180,E1 -23319.055,E2 -23319.055} C_VEL
LIN {X 0,Y 168.105,Z 429.507,A -85,B 0,C 180,E1 -23322.065,E2 -23322.065} C_VEL
LIN {X 0,Y 165.72,Z 437.88,A -85,B 0,C 180,E1 -23326.001,E2 -23326.001} C_VEL
LIN {X 0,Y 163.906,Z 444.51,A -85,B 0,C 180,E1 -23330.061,E2 -23330.061} C_VEL
LIN {X 0,Y 162.837,Z 449.184,A -85,B 0,C 180,E1 -23333.831,E2 -23333.831} C_VEL
LIN {X 0,Y 162.087,Z 452.287,A -85,B 0,C 180,E1 -23337.082,E2 -23337.082} C_VEL
LIN {X 0,Y 161.523,Z 455.227,A -85,B 0,C 180,E1 -23341.474,E2 -23341.474} C_VEL
LIN {X 0,Y 161.557,Z 456.463,A -85,B 0,C 180,E1 -23344.437,E2 -23344.437} C_VEL
LIN {X 0,Y 162.081,Z 457.283,A -85,B 0,C 180,E1 -23348.721,E2 -23348.721} C_VEL
LIN {X 0,Y 163.419,Z 456.817,A -85,B 0,C 180,E1 -23353.478,E2 -23353.478} C_VEL
LIN {X 0,Y 165.03,Z 455.473,A -85,B 0,C 180,E1 -23357.071,E2 -23357.071} C_VEL
LIN {X 0,Y 167.385,Z 452.929,A -85,B 0,C 180,E1 -23360.984,E2 -23360.984} C_VEL
LIN {X 0,Y 170.909,Z 448.567,A -85,B 0,C 180,E1 -23365.326,E2 -23365.326} C_VEL
LIN {X 0,Y 173.963,Z 444.418,A -85,B 0,C 180,E1 -23368.336,E2 -23368.336} C_VEL
LIN {X 0,Y 178.295,Z 438.116,A -85,B 0,C 180,E1 -23371.786,E2 -23371.786} C_VEL
LIN {X 0,Y 183.145,Z 430.242,A -85,B 0,C 180,E1 -23375.047,E2 -23375.047} C_VEL
LIN {X 0,Y 187.634,Z 422.003,A -85,B 0,C 180,E1 -23377.647,E2 -23377.647} C_VEL
LIN {X 0,Y 191.849,Z 413.221,A -85,B 0,C 180,E1 -23379.833,E2 -23379.833} C_VEL
LIN {X 0,Y 196.166,Z 402.861,A -85,B 0,C 180,E1 -23381.863,E2 -23381.863} C_VEL
LIN {X 0,Y 199.959,Z 392.06,A -85,B 0,C 180,E1 -23383.509,E2 -23383.509} C_VEL
LIN {X 0,Y 203.472,Z 379.649,A -85,B 0,C 180,E1 -23384.918,E2 -23384.918} C_VEL
LIN {X 0,Y 206.275,Z 366.24,A -85,B 0,C 180,E1 -23386.026,E2 -23386.026} C_VEL
LIN {X 0,Y 208.121,Z 353.3,A -85,B 0,C 180,E1 -23386.712,E2 -23386.712} C_VEL
LIN {X 0,Y 211.251,Z 317.077,A -85,B 0,C 180,E1 -23387.949,E2 -23387.949} C_VEL
LIN {X 0,Y 207.578,Z 309.066,A -85,B 0,C 180,E1 -23390.021,E2 -23390.021} C_VEL
LIN {X 0,Y 203.598,Z 302.089,A -85,B 0,C 180,E1 -23392.427,E2 -23392.427} C_VEL
LIN {X 0,Y 199.454,Z 295.243,A -85,B 0,C 180,E1 -23395.3,E2 -23395.3} C_VEL
LIN {X 0,Y 197.388,Z 292.173,A -85,B 0,C 180,E1 -23396.886,E2 -23396.886} C_VEL
LIN {X 0,Y 194.302,Z 287.573,A -85,B 0,C 180,E1 -23399.641,E2 -23399.641} C_VEL
LIN {X 0,Y 191.949,Z 284.126,A -85,B 0,C 180,E1 -23402.11,E2 -23402.11} C_VEL
LIN {X 0,Y 191.304,Z 283.18,A -85,B 0,C 180,E1 -23402.907,E2 -23402.907} C_VEL
LIN {X 0,Y 188.632,Z 280.641,A -85,B 0,C 180,E1 -23406.568,E2 -23406.568} C_VEL
LIN {X 0,Y 187.713,Z 278.321,A -85,B 0,C 180,E1 -23408.625,E2 -23408.625} C_VEL
LIN {X 0,Y 185.832,Z 277.48,A -85,B 0,C 180,E1 -23415.363,E2 -23415.363} C_VEL
LIN {X 0,Y 186.901,Z 278.14,A -85,B 0,C 180,E1 -23422.1,E2 -23422.1} C_VEL
LIN {X 0,Y 187.985,Z 279.996,A -85,B 0,C 180,E1 -23424.783,E2 -23424.783} C_VEL
LIN {X 0,Y 190.058,Z 283.409,A -85,B 0,C 180,E1 -23428.244,E2 -23428.244} C_VEL
LIN {X 0,Y 192.202,Z 286.502,A -85,B 0,C 180,E1 -23430.922,E2 -23430.922} C_VEL
LIN {X 0,Y 195.56,Z 292.199,A -85,B 0,C 180,E1 -23434.34,E2 -23434.34} C_VEL
LIN {X 0,Y 198.898,Z 298.21,A -85,B 0,C 180,E1 -23437.125,E2 -23437.125} C_VEL
LIN {X 0,Y 201.972,Z 304.173,A -85,B 0,C 180,E1 -23439.392,E2 -23439.392} C_VEL
LIN {X 0,Y 205.581,Z 311.758,A -85,B 0,C 180,E1 -23441.756,E2 -23441.756} C_VEL
LIN {X 0,Y 208.655,Z 319.355,A -85,B 0,C 180,E1 -23443.646,E2 -23443.646} C_VEL
LIN {X 0,Y 210.665,Z 325.321,A -85,B 0,C 180,E1 -23444.844,E2 -23444.844} C_VEL
LIN {X 0,Y 207.251,Z 364.621,A -85,B 0,C 180,E1 -23446.235,E2 -23446.235} C_VEL
LIN {X 0,Y 205.169,Z 377.28,A -85,B 0,C 180,E1 -23446.927,E2 -23446.927} C_VEL
LIN {X 0,Y 202.002,Z 390.444,A -85,B 0,C 180,E1 -23447.954,E2 -23447.954} C_VEL
LIN {X 0,Y 198.231,Z 402.707,A -85,B 0,C 180,E1 -23449.35,E2 -23449.35} C_VEL
LIN {X 0,Y 196.574,Z 407.309,A -85,B 0,C 180,E1 -23449.981,E2 -23449.981} C_VEL
LIN {X 0,Y 194.173,Z 412.366,A -85,B 0,C 180,E1 -23450.617,E2 -23450.617} C_VEL
LIN {X 0,Y 188.749,Z 420.29,A -85,B 0,C 180,E1 -23451.428,E2 -23451.428} C_VEL
LIN {X 0,Y 183.104,Z 427.652,A -85,B 0,C 180,E1 -23452.428,E2 -23452.428} C_VEL
LIN {X 0,Y 180.347,Z 431.835,A -85,B 0,C 180,E1 -23453.375,E2 -23453.375} C_VEL
LIN {X 0,Y 174.914,Z 441.259,A -85,B 0,C 180,E1 -23456.464,E2 -23456.464} C_VEL
LIN {X 0,Y 170.092,Z 448.621,A -85,B 0,C 180,E1 -23459.593,E2 -23459.593} C_VEL
LIN {X 0,Y 166.049,Z 454.598,A -85,B 0,C 180,E1 -23462.964,E2 -23462.964} C_VEL
LIN {X 0,Y 161.975,Z 460.006,A -85,B 0,C 180,E1 -23467.015,E2 -23467.015} C_VEL
LIN {X 0,Y 158.329,Z 464.446,A -85,B 0,C 180,E1 -23471.898,E2 -23471.898} C_VEL
LIN {X 0,Y 157.008,Z 466.058,A -85,B 0,C 180,E1 -23474.421,E2 -23474.421} C_VEL
LIN {X 0,Y 156.055,Z 467.258,A -85,B 0,C 180,E1 -23476.987,E2 -23476.987} C_VEL
LIN {X 0,Y 154.934,Z 468.46,A -85,B 0,C 180,E1 -23482.179,E2 -23482.179} C_VEL
LIN {X 0,Y 154.774,Z 468.495,A -85,B 0,C 180,E1 -23484.79,E2 -23484.79} C_VEL
LIN {X 0,Y 154.778,Z 468.078,A -85,B 0,C 180,E1 -23487.639,E2 -23487.639} C_VEL
LIN {X 0,Y 154.942,Z 467.348,A -85,B 0,C 180,E1 -23490,E2 -23490} C_VEL
LIN {X 0,Y 154.844,Z 465.961,A -85,B 0,C 180,E1 -23492.894,E2 -23492.894} C_VEL
LIN {X 0,Y 154.92,Z 463.464,A -85,B 0,C 180,E1 -23496.512,E2 -23496.512} C_VEL
LIN {X 0,Y 155.418,Z 459.739,A -85,B 0,C 180,E1 -23500.421,E2 -23500.421} C_VEL
LIN {X 0,Y 156.361,Z 454.839,A -85,B 0,C 180,E1 -23504.312,E2 -23504.312} C_VEL
LIN {X 0,Y 158.05,Z 448.642,A -85,B 0,C 180,E1 -23508.135,E2 -23508.135} C_VEL
LIN {X 0,Y 160.367,Z 440.902,A -85,B 0,C 180,E1 -23511.87,E2 -23511.87} C_VEL
LIN {X 0,Y 162.407,Z 433.732,A -85,B 0,C 180,E1 -23514.64,E2 -23514.64} C_VEL
LIN {X 0,Y 165.056,Z 424.251,A -85,B 0,C 180,E1 -23517.584,E2 -23517.584} C_VEL
LIN {X 0,Y 167.211,Z 416.261,A -85,B 0,C 180,E1 -23519.594,E2 -23519.594} C_VEL
LIN {X 0,Y 170.132,Z 405.171,A -85,B 0,C 180,E1 -23521.781,E2 -23521.781} C_VEL
LIN {X 0,Y 172.369,Z 394.733,A -85,B 0,C 180,E1 -23523.396,E2 -23523.396} C_VEL
LIN {X 0,Y 174.589,Z 382.365,A -85,B 0,C 180,E1 -23524.827,E2 -23524.827} C_VEL
LIN {X 0,Y 176.25,Z 369.697,A -85,B 0,C 180,E1 -23525.849,E2 -23525.849} C_VEL
LIN {X 0,Y 177.376,Z 354.694,A -85,B 0,C 180,E1 -23526.586,E2 -23526.586} C_VEL
LIN {X 0,Y 179.4,Z 318.876,A -85,B 0,C 180,E1 -23528.051,E2 -23528.051} C_VEL
LIN {X 0,Y 177.662,Z 303.077,A -85,B 0,C 180,E1 -23529.184,E2 -23529.184} C_VEL
LIN {X 0,Y 170.632,Z 284.062,A -85,B 0,C 180,E1 -23531.641,E2 -23531.641} C_VEL
LIN {X 0,Y 164.931,Z 271.212,A -85,B 0,C 180,E1 -23533.675,E2 -23533.675} C_VEL
LIN {X 0,Y 159.121,Z 259.509,A -85,B 0,C 180,E1 -23535.836,E2 -23535.836} C_VEL
LIN {X 0,Y 157.471,Z 256.046,A -85,B 0,C 180,E1 -23536.545,E2 -23536.545} C_VEL
LIN {X 0,Y 157.202,Z 254.903,A -85,B 0,C 180,E1 -23537.358,E2 -23537.358} C_VEL
LIN {X 0,Y 157.275,Z 254.893,A -85,B 0,C 180,E1 -23543.546,E2 -23543.546} C_VEL
LIN {X 0,Y 157.288,Z 254.889,A -85,B 0,C 180,E1 -23548.097,E2 -23548.097} C_VEL
LIN {X 0,Y 157.279,Z 254.887,A -85,B 0,C 180,E1 -23553.444,E2 -23553.444} C_VEL
LIN {X 0,Y 157.368,Z 254.86,A -85,B 0,C 180,E1 -23559.69,E2 -23559.69} C_VEL
LIN {X 0,Y 157.417,Z 254.85,A -85,B 0,C 180,E1 -23564.448,E2 -23564.448} C_VEL
LIN {X 0,Y 157.688,Z 254.841,A -85,B 0,C 180,E1 -23569.717,E2 -23569.717} C_VEL
LIN {X 0,Y 157.753,Z 254.817,A -85,B 0,C 180,E1 -23572.305,E2 -23572.305} C_VEL
LIN {X 0,Y 158.221,Z 254.747,A -85,B 0,C 180,E1 -23579.986,E2 -23579.986} C_VEL
LIN {X 0,Y 157.747,Z 254.827,A -85,B 0,C 180,E1 -23587.666,E2 -23587.666} C_VEL
LIN {X 0,Y 157.621,Z 254.841,A -85,B 0,C 180,E1 -23591.213,E2 -23591.213} C_VEL
LIN {X 0,Y 157.421,Z 254.872,A -85,B 0,C 180,E1 -23595.521,E2 -23595.521} C_VEL
LIN {X 0,Y 157.348,Z 254.878,A -85,B 0,C 180,E1 -23600.919,E2 -23600.919} C_VEL
LIN {X 0,Y 157.287,Z 254.875,A -85,B 0,C 180,E1 -23606.667,E2 -23606.667} C_VEL
LIN {X 0,Y 157.238,Z 254.842,A -85,B 0,C 180,E1 -23612.417,E2 -23612.417} C_VEL
LIN {X 0,Y 157.228,Z 254.886,A -85,B 0,C 180,E1 -23616.431,E2 -23616.431} C_VEL
LIN {X 0,Y 157.157,Z 254.902,A -85,B 0,C 180,E1 -23622.106,E2 -23622.106} C_VEL
LIN {X 0,Y 157.155,Z 254.908,A -85,B 0,C 180,E1 -23627.872,E2 -23627.872} C_VEL
LIN {X 0,Y 157.227,Z 254.903,A -85,B 0,C 180,E1 -23633.542,E2 -23633.542} C_VEL
LIN {X 0,Y 157.251,Z 254.897,A -85,B 0,C 180,E1 -23638.088,E2 -23638.088} C_VEL
LIN {X 0,Y 157.282,Z 254.893,A -85,B 0,C 180,E1 -23643.459,E2 -23643.459} C_VEL
LIN {X 0,Y 157.402,Z 254.886,A -85,B 0,C 180,E1 -23649.61,E2 -23649.61} C_VEL
LIN {X 0,Y 157.468,Z 254.868,A -85,B 0,C 180,E1 -23655.79,E2 -23655.79} C_VEL
LIN {X 0,Y 157.538,Z 254.993,A -85,B 0,C 180,E1 -23657.112,E2 -23657.112} C_VEL
LIN {X 0,Y 158.604,Z 257.795,A -85,B 0,C 180,E1 -23657.577,E2 -23657.577} C_VEL
LIN {X 0,Y 160.226,Z 260.048,A -85,B 0,C 180,E1 -23658.148,E2 -23658.148} C_VEL
LIN {X 0,Y 165.839,Z 269.548,A -85,B 0,C 180,E1 -23660.107,E2 -23660.107} C_VEL
LIN {X 0,Y 174.617,Z 285.983,A -85,B 0,C 180,E1 -23662.971,E2 -23662.971} C_VEL
LIN {X 0,Y 178.659,Z 296.084,A -85,B 0,C 180,E1 -23664.306,E2 -23664.306} C_VEL
LIN {X 0,Y 180.356,Z 300.538,A -85,B 0,C 180,E1 -23664.855,E2 -23664.855} C_VEL
LIN {X 0,Y 176.992,Z 354.318,A -85,B 0,C 180,E1 -23667.07,E2 -23667.07} C_VEL
LIN {X 0,Y 175.517,Z 367.293,A -85,B 0,C 180,E1 -23668.008,E2 -23668.008} C_VEL
LIN {X 0,Y 173.738,Z 379.767,A -85,B 0,C 180,E1 -23669.362,E2 -23669.362} C_VEL
LIN {X 0,Y 171.344,Z 392.019,A -85,B 0,C 180,E1 -23671.175,E2 -23671.175} C_VEL
LIN {X 0,Y 168.654,Z 403.517,A -85,B 0,C 180,E1 -23673.408,E2 -23673.408} C_VEL
LIN {X 0,Y 165.838,Z 414.168,A -85,B 0,C 180,E1 -23676.081,E2 -23676.081} C_VEL
LIN {X 0,Y 162.918,Z 423.815,A -85,B 0,C 180,E1 -23679.17,E2 -23679.17} C_VEL
LIN {X 0,Y 160.44,Z 432.335,A -85,B 0,C 180,E1 -23682.651,E2 -23682.651} C_VEL
LIN {X 0,Y 158.444,Z 439.017,A -85,B 0,C 180,E1 -23686.094,E2 -23686.094} C_VEL
LIN {X 0,Y 156.847,Z 444.76,A -85,B 0,C 180,E1 -23689.838,E2 -23689.838} C_VEL
LIN {X 0,Y 155.69,Z 449.629,A -85,B 0,C 180,E1 -23693.97,E2 -23693.97} C_VEL
LIN {X 0,Y 154.753,Z 453.499,A -85,B 0,C 180,E1 -23698.479,E2 -23698.479} C_VEL
LIN {X 0,Y 154.395,Z 456.098,A -85,B 0,C 180,E1 -23703.108,E2 -23703.108} C_VEL
LIN {X 0,Y 154.581,Z 457.106,A -85,B 0,C 180,E1 -23706.23,E2 -23706.23} C_VEL
LIN {X 0,Y 155.16,Z 457.584,A -85,B 0,C 180,E1 -23709.672,E2 -23709.672} C_VEL
LIN {X 0,Y 156.525,Z 457.154,A -85,B 0,C 180,E1 -23714.102,E2 -23714.102} C_VEL
LIN {X 0,Y 158.788,Z 455.361,A -85,B 0,C 180,E1 -23718.799,E2 -23718.799} C_VEL
LIN {X 0,Y 162.004,Z 452.025,A -85,B 0,C 180,E1 -23723.564,E2 -23723.564} C_VEL
LIN {X 0,Y 165.967,Z 447.329,A -85,B 0,C 180,E1 -23727.875,E2 -23727.875} C_VEL
LIN {X 0,Y 170.121,Z 441.951,A -85,B 0,C 180,E1 -23731.384,E2 -23731.384} C_VEL
LIN {X 0,Y 174.832,Z 435.12,A -85,B 0,C 180,E1 -23734.745,E2 -23734.745} C_VEL
LIN {X 0,Y 179.471,Z 427.682,A -85,B 0,C 180,E1 -23737.56,E2 -23737.56} C_VEL
LIN {X 0,Y 184.623,Z 418.291,A -85,B 0,C 180,E1 -23740.293,E2 -23740.293} C_VEL
LIN {X 0,Y 189.517,Z 407.974,A -85,B 0,C 180,E1 -23742.572,E2 -23742.572} C_VEL
LIN {X 0,Y 193.465,Z 398.081,A -85,B 0,C 180,E1 -23744.289,E2 -23744.289} C_VEL
LIN {X 0,Y 197.341,Z 386.517,A -85,B 0,C 180,E1 -23745.822,E2 -23745.822} C_VEL
LIN {X 0,Y 200.442,Z 374.411,A -85,B 0,C 180,E1 -23747.031,E2 -23747.031} C_VEL
LIN {X 0,Y 202.896,Z 361.656,A -85,B 0,C 180,E1 -23747.916,E2 -23747.916} C_VEL
LIN {X 0,Y 204.495,Z 348.526,A -85,B 0,C 180,E1 -23748.497,E2 -23748.497} C_VEL
LIN {X 0,Y 207.015,Z 320.014,A -85,B 0,C 180,E1 -23749.468,E2 -23749.468} C_VEL
LIN {X 0,Y 204.205,Z 313.813,A -85,B 0,C 180,E1 -23751.204,E2 -23751.204} C_VEL
LIN {X 0,Y 199.882,Z 305.916,A -85,B 0,C 180,E1 -23754.068,E2 -23754.068} C_VEL
LIN {X 0,Y 195.756,Z 299.005,A -85,B 0,C 180,E1 -23757.265,E2 -23757.265} C_VEL
LIN {X 0,Y 192.89,Z 294.659,A -85,B 0,C 180,E1 -23759.918,E2 -23759.918} C_VEL
LIN {X 0,Y 190.167,Z 290.327,A -85,B 0,C 180,E1 -23762.998,E2 -23762.998} C_VEL
LIN {X 0,Y 187.26,Z 287.332,A -85,B 0,C 180,E1 -23767.167,E2 -23767.167} C_VEL
LIN {X 0,Y 186.348,Z 285.15,A -85,B 0,C 180,E1 -23769.391,E2 -23769.391} C_VEL
LIN {X 0,Y 184.827,Z 284.511,A -85,B 0,C 180,E1 -23775.449,E2 -23775.449} C_VEL
LIN {X 0,Y 185.833,Z 285.147,A -85,B 0,C 180,E1 -23781.93,E2 -23781.93} C_VEL
LIN {X 0,Y 186.801,Z 286.97,A -85,B 0,C 180,E1 -23784.459,E2 -23784.459} C_VEL
LIN {X 0,Y 188.69,Z 290.243,A -85,B 0,C 180,E1 -23787.808,E2 -23787.808} C_VEL
LIN {X 0,Y 190.504,Z 293.063,A -85,B 0,C 180,E1 -23790.254,E2 -23790.254} C_VEL
LIN {X 0,Y 193.55,Z 298.468,A -85,B 0,C 180,E1 -23793.543,E2 -23793.543} C_VEL
LIN {X 0,Y 196.656,Z 304.423,A -85,B 0,C 180,E1 -23796.338,E2 -23796.338} C_VEL
LIN {X 0,Y 199.931,Z 311.144,A -85,B 0,C 180,E1 -23798.905,E2 -23798.905} C_VEL
LIN {X 0,Y 203.203,Z 318.628,A -85,B 0,C 180,E1 -23801.169,E2 -23801.169} C_VEL
LIN {X 0,Y 205.898,Z 326.031,A -85,B 0,C 180,E1 -23802.964,E2 -23802.964} C_VEL
LIN {X 0,Y 206.427,Z 327.905,A -85,B 0,C 180,E1 -23803.327,E2 -23803.327} C_VEL
LIN {X 0,Y 203.157,Z 364.079,A -85,B 0,C 180,E1 -23804.609,E2 -23804.609} C_VEL
LIN {X 0,Y 200.939,Z 377.077,A -85,B 0,C 180,E1 -23805.31,E2 -23805.31} C_VEL
LIN {X 0,Y 197.762,Z 389.931,A -85,B 0,C 180,E1 -23806.311,E2 -23806.311} C_VEL
LIN {X 0,Y 194.083,Z 401.496,A -85,B 0,C 180,E1 -23807.591,E2 -23807.591} C_VEL
LIN {X 0,Y 189.698,Z 412.737,A -85,B 0,C 180,E1 -23809.235,E2 -23809.235} C_VEL
LIN {X 0,Y 185.07,Z 422.948,A -85,B 0,C 180,E1 -23811.203,E2 -23811.203} C_VEL
LIN {X 0,Y 180.347,Z 431.835,A -85,B 0,C 180,E1 -23813.375,E2 -23813.375} C_VEL
LIN {X 0,Y 177.547,Z 435.915,A -85,B 0,C 180,E1 -23814.418,E2 -23814.418} C_VEL
LIN {X 0,Y 171.486,Z 442.175,A -85,B 0,C 180,E1 -23815.989,E2 -23815.989} C_VEL
LIN {X 0,Y 165.435,Z 447.822,A -85,B 0,C 180,E1 -23817.841,E2 -23817.841} C_VEL
LIN {X 0,Y 162.714,Z 450.872,A -85,B 0,C 180,E1 -23819.315,E2 -23819.315} C_VEL
LIN {X 0,Y 157.832,Z 457.318,A -85,B 0,C 180,E1 -23823.56,E2 -23823.56} C_VEL
LIN {X 0,Y 154.423,Z 461.4,A -85,B 0,C 180,E1 -23827.242,E2 -23827.242} C_VEL
LIN {X 0,Y 151.594,Z 464.467,A -85,B 0,C 180,E1 -23831.064,E2 -23831.064} C_VEL
LIN {X 0,Y 150.144,Z 466.004,A -85,B 0,C 180,E1 -23833.69,E2 -23833.69} C_VEL
LIN {X 0,Y 148.354,Z 467.855,A -85,B 0,C 180,E1 -23839.077,E2 -23839.077} C_VEL
LIN {X 0,Y 147.706,Z 468.204,A -85,B 0,C 180,E1 -23844.54,E2 -23844.54} C_VEL
LIN {X 0,Y 147.707,Z 467.562,A -85,B 0,C 180,E1 -23848.023,E2 -23848.023} C_VEL
LIN {X 0,Y 147.876,Z 466.919,A -85,B 0,C 180,E1 -23850,E2 -23850} C_VEL
LIN {X 0,Y 147.756,Z 465.644,A -85,B 0,C 180,E1 -23852.726,E2 -23852.726} C_VEL
LIN {X 0,Y 147.874,Z 462.885,A -85,B 0,C 180,E1 -23856.824,E2 -23856.824} C_VEL
LIN {X 0,Y 148.392,Z 459.049,A -85,B 0,C 180,E1 -23860.92,E2 -23860.92} C_VEL
LIN {X 0,Y 149.44,Z 454.032,A -85,B 0,C 180,E1 -23864.99,E2 -23864.99} C_VEL
LIN {X 0,Y 151.273,Z 447.709,A -85,B 0,C 180,E1 -23868.978,E2 -23868.978} C_VEL
LIN {X 0,Y 153.753,Z 439.752,A -85,B 0,C 180,E1 -23872.863,E2 -23872.863} C_VEL
LIN {X 0,Y 155.7,Z 433.242,A -85,B 0,C 180,E1 -23875.45,E2 -23875.45} C_VEL
LIN {X 0,Y 158.807,Z 422.721,A -85,B 0,C 180,E1 -23878.768,E2 -23878.768} C_VEL
LIN {X 0,Y 161.414,Z 413.174,A -85,B 0,C 180,E1 -23881.133,E2 -23881.133} C_VEL
LIN {X 0,Y 164.435,Z 401.398,A -85,B 0,C 180,E1 -23883.385,E2 -23883.385} C_VEL
LIN {X 0,Y 167.118,Z 388.895,A -85,B 0,C 180,E1 -23885.142,E2 -23885.142} C_VEL
LIN {X 0,Y 169.194,Z 375.821,A -85,B 0,C 180,E1 -23886.477,E2 -23886.477} C_VEL
LIN {X 0,Y 170.632,Z 362.95,A -85,B 0,C 180,E1 -23887.317,E2 -23887.317} C_VEL
LIN {X 0,Y 173.199,Z 319.113,A -85,B 0,C 180,E1 -23889.199,E2 -23889.199} C_VEL
LIN {X 0,Y 171.687,Z 305.273,A -85,B 0,C 180,E1 -23890.247,E2 -23890.247} C_VEL
LIN {X 0,Y 164.942,Z 286.842,A -85,B 0,C 180,E1 -23892.768,E2 -23892.768} C_VEL
LIN {X 0,Y 158.806,Z 272.953,A -85,B 0,C 180,E1 -23895.087,E2 -23895.087} C_VEL
LIN {X 0,Y 153.876,Z 263.127,A -85,B 0,C 180,E1 -23897.052,E2 -23897.052} C_VEL
LIN {X 0,Y 152.094,Z 259.828,A -85,B 0,C 180,E1 -23897.791,E2 -23897.791} C_VEL
LIN {X 0,Y 150.496,Z 257.254,A -85,B 0,C 180,E1 -23898.437,E2 -23898.437} C_VEL
LIN {X 0,Y 150.161,Z 255.781,A -85,B 0,C 180,E1 -23898.714,E2 -23898.714} C_VEL
LIN {X 0,Y 150.193,Z 255.778,A -85,B 0,C 180,E1 -23902.699,E2 -23902.699} C_VEL
LIN {X 0,Y 150.216,Z 255.773,A -85,B 0,C 180,E1 -23907.365,E2 -23907.365} C_VEL
LIN {X 0,Y 150.194,Z 255.77,A -85,B 0,C 180,E1 -23912.753,E2 -23912.753} C_VEL
LIN {X 0,Y 150.291,Z 255.745,A -85,B 0,C 180,E1 -23919.265,E2 -23919.265} C_VEL
LIN {X 0,Y 150.322,Z 255.725,A -85,B 0,C 180,E1 -23923.694,E2 -23923.694} C_VEL
LIN {X 0,Y 150.608,Z 255.725,A -85,B 0,C 180,E1 -23929.228,E2 -23929.228} C_VEL
LIN {X 0,Y 150.677,Z 255.702,A -85,B 0,C 180,E1 -23931.942,E2 -23931.942} C_VEL
LIN {X 0,Y 151.181,Z 255.623,A -85,B 0,C 180,E1 -23939.985,E2 -23939.985} C_VEL
LIN {X 0,Y 150.67,Z 255.706,A -85,B 0,C 180,E1 -23948.028,E2 -23948.028} C_VEL
LIN {X 0,Y 150.562,Z 255.721,A -85,B 0,C 180,E1 -23951.414,E2 -23951.414} C_VEL
LIN {X 0,Y 150.333,Z 255.753,A -85,B 0,C 180,E1 -23956.273,E2 -23956.273} C_VEL
LIN {X 0,Y 150.331,Z 255.751,A -85,B 0,C 180,E1 -23960.775,E2 -23960.775} C_VEL
LIN {X 0,Y 150.216,Z 255.75,A -85,B 0,C 180,E1 -23967.263,E2 -23967.263} C_VEL
LIN {X 0,Y 150.178,Z 255.72,A -85,B 0,C 180,E1 -23972.612,E2 -23972.612} C_VEL
LIN {X 0,Y 150.139,Z 255.775,A -85,B 0,C 180,E1 -23977.462,E2 -23977.462} C_VEL
LIN {X 0,Y 150.1,Z 255.783,A -85,B 0,C 180,E1 -23981.484,E2 -23981.484} C_VEL
LIN {X 0,Y 150.091,Z 255.784,A -85,B 0,C 180,E1 -23985.384,E2 -23985.384} C_VEL
LIN {X 0,Y 150.103,Z 255.781,A -85,B 0,C 180,E1 -23989.044,E2 -23989.044} C_VEL
LIN {X 0,Y 150.14,Z 255.782,A -85,B 0,C 180,E1 -23992.698,E2 -23992.698} C_VEL
LIN {X 0,Y 150.173,Z 255.774,A -85,B 0,C 180,E1 -23997.36,E2 -23997.36} C_VEL
LIN {X 0,Y 150.203,Z 255.772,A -85,B 0,C 180,E1 -24002.709,E2 -24002.709} C_VEL
LIN {X 0,Y 150.345,Z 255.763,A -85,B 0,C 180,E1 -24009.163,E2 -24009.163} C_VEL
LIN {X 0,Y 150.409,Z 255.751,A -85,B 0,C 180,E1 -24015.056,E2 -24015.056} C_VEL
LIN {X 0,Y 151.396,Z 258.551,A -85,B 0,C 180,E1 -24015.589,E2 -24015.589} C_VEL
LIN {X 0,Y 153.163,Z 261.009,A -85,B 0,C 180,E1 -24016.27,E2 -24016.27} C_VEL
LIN {X 0,Y 159.395,Z 271.189,A -85,B 0,C 180,E1 -24018.621,E2 -24018.621} C_VEL
LIN {X 0,Y 169.38,Z 289.96,A -85,B 0,C 180,E1 -24022.076,E2 -24022.076} C_VEL
LIN {X 0,Y 174.06,Z 301.997,A -85,B 0,C 180,E1 -24023.718,E2 -24023.718} C_VEL
LIN {X 0,Y 170.799,Z 354.118,A -85,B 0,C 180,E1 -24025.941,E2 -24025.941} C_VEL
LIN {X 0,Y 169.313,Z 366.546,A -85,B 0,C 180,E1 -24026.833,E2 -24026.833} C_VEL
LIN {X 0,Y 167.535,Z 378.991,A -85,B 0,C 180,E1 -24028.197,E2 -24028.197} C_VEL
LIN {X 0,Y 165.105,Z 391.197,A -85,B 0,C 180,E1 -24030,E2 -24030} C_VEL
LIN {X 0,Y 162.437,Z 402.303,A -85,B 0,C 180,E1 -24032.169,E2 -24032.169} C_VEL
LIN {X 0,Y 159.658,Z 412.593,A -85,B 0,C 180,E1 -24034.742,E2 -24034.742} C_VEL
LIN {X 0,Y 156.754,Z 422.074,A -85,B 0,C 180,E1 -24037.73,E2 -24037.73} C_VEL
LIN {X 0,Y 154.145,Z 430.594,A -85,B 0,C 180,E1 -24041.173,E2 -24041.173} C_VEL
LIN {X 0,Y 151.764,Z 438.246,A -85,B 0,C 180,E1 -24045.096,E2 -24045.096} C_VEL
LIN {X 0,Y 149.933,Z 444.425,A -85,B 0,C 180,E1 -24049.154,E2 -24049.154} C_VEL
LIN {X 0,Y 148.625,Z 449.676,A -85,B 0,C 180,E1 -24053.699,E2 -24053.699} C_VEL
LIN {X 0,Y 147.648,Z 453.61,A -85,B 0,C 180,E1 -24058.423,E2 -24058.423} C_VEL
LIN {X 0,Y 147.322,Z 455.545,A -85,B 0,C 180,E1 -24061.65,E2 -24061.65} C_VEL
LIN {X 0,Y 147.459,Z 457.174,A -85,B 0,C 180,E1 -24065.912,E2 -24065.912} C_VEL
LIN {X 0,Y 148.274,Z 457.868,A -85,B 0,C 180,E1 -24070.706,E2 -24070.706} C_VEL
LIN {X 0,Y 149.837,Z 457.363,A -85,B 0,C 180,E1 -24075.311,E2 -24075.311} C_VEL
LIN {X 0,Y 152.095,Z 455.76,A -85,B 0,C 180,E1 -24079.713,E2 -24079.713} C_VEL
LIN {X 0,Y 155.41,Z 452.624,A -85,B 0,C 180,E1 -24084.486,E2 -24084.486} C_VEL
LIN {X 0,Y 159.792,Z 447.859,A -85,B 0,C 180,E1 -24089.135,E2 -24089.135} C_VEL
LIN {X 0,Y 165.081,Z 441.438,A -85,B 0,C 180,E1 -24093.381,E2 -24093.381} C_VEL
LIN {X 0,Y 170.161,Z 434.469,A -85,B 0,C 180,E1 -24096.772,E2 -24096.772} C_VEL
LIN {X 0,Y 175.801,Z 425.652,A -85,B 0,C 180,E1 -24099.956,E2 -24099.956} C_VEL
LIN {X 0,Y 181.044,Z 416.256,A -85,B 0,C 180,E1 -24102.531,E2 -24102.531} C_VEL
LIN {X 0,Y 185.897,Z 406.112,A -85,B 0,C 180,E1 -24104.668,E2 -24104.668} C_VEL
LIN {X 0,Y 190.525,Z 394.47,A -85,B 0,C 180,E1 -24106.535,E2 -24106.535} C_VEL
LIN {X 0,Y 194.446,Z 382.362,A -85,B 0,C 180,E1 -24107.99,E2 -24107.99} C_VEL
LIN {X 0,Y 197.493,Z 369.798,A -85,B 0,C 180,E1 -24109.09,E2 -24109.09} C_VEL
LIN {X 0,Y 199.549,Z 358.106,A -85,B 0,C 180,E1 -24109.789,E2 -24109.789} C_VEL
LIN {X 0,Y 201.695,Z 337.132,A -85,B 0,C 180,E1 -24110.579,E2 -24110.579} C_VEL
LIN {X 0,Y 202.963,Z 323.043,A -85,B 0,C 180,E1 -24111.072,E2 -24111.072} C_VEL
LIN {X 0,Y 200.465,Z 317.632,A -85,B 0,C 180,E1 -24112.735,E2 -24112.735} C_VEL
LIN {X 0,Y 196.962,Z 311.105,A -85,B 0,C 180,E1 -24115.296,E2 -24115.296} C_VEL
LIN {X 0,Y 193.58,Z 305.173,A -85,B 0,C 180,E1 -24118.138,E2 -24118.138} C_VEL
LIN {X 0,Y 190.343,Z 300.129,A -85,B 0,C 180,E1 -24121.39,E2 -24121.39} C_VEL
LIN {X 0,Y 188.362,Z 296.781,A -85,B 0,C 180,E1 -24123.935,E2 -24123.935} C_VEL
LIN {X 0,Y 186.011,Z 294.168,A -85,B 0,C 180,E1 -24127.612,E2 -24127.612} C_VEL
LIN {X 0,Y 185.281,Z 292.152,A -85,B 0,C 180,E1 -24129.533,E2 -24129.533} C_VEL
LIN {X 0,Y 183.838,Z 291.58,A -85,B 0,C 180,E1 -24137.117,E2 -24137.117} C_VEL
LIN {X 0,Y 184.859,Z 292.348,A -85,B 0,C 180,E1 -24142.052,E2 -24142.052} C_VEL
LIN {X 0,Y 185.565,Z 293.78,A -85,B 0,C 180,E1 -24143.979,E2 -24143.979} C_VEL
LIN {X 0,Y 187.215,Z 296.859,A -85,B 0,C 180,E1 -24147.175,E2 -24147.175} C_VEL
LIN {X 0,Y 188.831,Z 299.507,A -85,B 0,C 180,E1 -24149.505,E2 -24149.505} C_VEL
LIN {X 0,Y 191.71,Z 305.033,A -85,B 0,C 180,E1 -24152.875,E2 -24152.875} C_VEL
LIN {X 0,Y 194.512,Z 310.73,A -85,B 0,C 180,E1 -24155.585,E2 -24155.585} C_VEL
LIN {X 0,Y 197.642,Z 317.609,A -85,B 0,C 180,E1 -24158.189,E2 -24158.189} C_VEL
LIN {X 0,Y 200.688,Z 325.211,A -85,B 0,C 180,E1 -24160.467,E2 -24160.467} C_VEL
LIN {X 0,Y 202.401,Z 330.291,A -85,B 0,C 180,E1 -24161.696,E2 -24161.696} C_VEL
LIN {X 0,Y 199.199,Z 364.131,A -85,B 0,C 180,E1 -24162.931,E2 -24162.931} C_VEL
LIN {X 0,Y 196.859,Z 377.111,A -85,B 0,C 180,E1 -24163.63,E2 -24163.63} C_VEL
LIN {X 0,Y 193.671,Z 389.488,A -85,B 0,C 180,E1 -24164.591,E2 -24164.591} C_VEL
LIN {X 0,Y 189.56,Z 401.82,A -85,B 0,C 180,E1 -24165.961,E2 -24165.961} C_VEL
LIN {X 0,Y 185.006,Z 412.959,A -85,B 0,C 180,E1 -24167.603,E2 -24167.603} C_VEL
LIN {X 0,Y 180.166,Z 423.094,A -85,B 0,C 180,E1 -24169.572,E2 -24169.572} C_VEL
LIN {X 0,Y 174.509,Z 433.106,A -85,B 0,C 180,E1 -24172.11,E2 -24172.11} C_VEL
LIN {X 0,Y 169.077,Z 441.924,A -85,B 0,C 180,E1 -24175.143,E2 -24175.143} C_VEL
LIN {X 0,Y 164.014,Z 449.096,A -85,B 0,C 180,E1 -24178.339,E2 -24178.339} C_VEL
LIN {X 0,Y 162.714,Z 450.872,A -85,B 0,C 180,E1 -24179.315,E2 -24179.315} C_VEL
LIN {X 0,Y 160.055,Z 453.738,A -85,B 0,C 180,E1 -24180.895,E2 -24180.895} C_VEL
LIN {X 0,Y 154.235,Z 457.924,A -85,B 0,C 180,E1 -24183.392,E2 -24183.392} C_VEL
LIN {X 0,Y 148.588,Z 461.409,A -85,B 0,C 180,E1 -24186.182,E2 -24186.182} C_VEL
LIN {X 0,Y 146.278,Z 463.092,A -85,B 0,C 180,E1 -24188.188,E2 -24188.188} C_VEL
LIN {X 0,Y 143.31,Z 465.918,A -85,B 0,C 180,E1 -24192.889,E2 -24192.889} C_VEL
LIN {X 0,Y 141.373,Z 467.667,A -85,B 0,C 180,E1 -24198.531,E2 -24198.531} C_VEL
LIN {X 0,Y 140.843,Z 467.977,A -85,B 0,C 180,E1 -24201.391,E2 -24201.391} C_VEL
LIN {X 0,Y 140.637,Z 467.875,A -85,B 0,C 180,E1 -24204.264,E2 -24204.264} C_VEL
LIN {X 0,Y 140.643,Z 467.038,A -85,B 0,C 180,E1 -24208.446,E2 -24208.446} C_VEL
LIN {X 0,Y 140.781,Z 466.482,A -85,B 0,C 180,E1 -24210,E2 -24210} C_VEL
LIN {X 0,Y 140.681,Z 465.161,A -85,B 0,C 180,E1 -24212.864,E2 -24212.864} C_VEL
LIN {X 0,Y 140.809,Z 462.301,A -85,B 0,C 180,E1 -24217.168,E2 -24217.168} C_VEL
LIN {X 0,Y 141.391,Z 458.359,A -85,B 0,C 180,E1 -24221.468,E2 -24221.468} C_VEL
LIN {X 0,Y 142.815,Z 452.223,A -85,B 0,C 180,E1 -24226.437,E2 -24226.437} C_VEL
LIN {X 0,Y 144.928,Z 445.483,A -85,B 0,C 180,E1 -24230.583,E2 -24230.583} C_VEL
LIN {X 0,Y 147.146,Z 438.589,A -85,B 0,C 180,E1 -24233.952,E2 -24233.952} C_VEL
LIN {X 0,Y 150.046,Z 429.569,A -85,B 0,C 180,E1 -24237.463,E2 -24237.463} C_VEL
LIN {X 0,Y 152.966,Z 420.083,A -85,B 0,C 180,E1 -24240.357,E2 -24240.357} C_VEL
LIN {X 0,Y 155.392,Z 411.383,A -85,B 0,C 180,E1 -24242.484,E2 -24242.484} C_VEL
LIN {X 0,Y 158.113,Z 400.806,A -85,B 0,C 180,E1 -24244.521,E2 -24244.521} C_VEL
LIN {X 0,Y 160.913,Z 388.22,A -85,B 0,C 180,E1 -24246.323,E2 -24246.323} C_VEL
LIN {X 0,Y 163.059,Z 374.991,A -85,B 0,C 180,E1 -24247.693,E2 -24247.693} C_VEL
LIN {X 0,Y 164.557,Z 361.843,A -85,B 0,C 180,E1 -24248.544,E2 -24248.544} C_VEL
LIN {X 0,Y 167.066,Z 319.865,A -85,B 0,C 180,E1 -24250.405,E2 -24250.405} C_VEL
LIN {X 0,Y 165.752,Z 307.416,A -85,B 0,C 180,E1 -24251.396,E2 -24251.396} C_VEL
LIN {X 0,Y 159.272,Z 289.647,A -85,B 0,C 180,E1 -24253.945,E2 -24253.945} C_VEL
LIN {X 0,Y 153.53,Z 276.499,A -85,B 0,C 180,E1 -24256.279,E2 -24256.279} C_VEL
LIN {X 0,Y 147.837,Z 264.983,A -85,B 0,C 180,E1 -24258.713,E2 -24258.713} C_VEL
LIN {X 0,Y 145.756,Z 261.655,A -85,B 0,C 180,E1 -24259.597,E2 -24259.597} C_VEL
LIN {X 0,Y 143.659,Z 258.765,A -85,B 0,C 180,E1 -24260.49,E2 -24260.49} C_VEL
LIN {X 0,Y 143.083,Z 256.663,A -85,B 0,C 180,E1 -24260.896,E2 -24260.896} C_VEL
LIN {X 0,Y 143.184,Z 256.649,A -85,B 0,C 180,E1 -24267.305,E2 -24267.305} C_VEL
LIN {X 0,Y 143.116,Z 256.651,A -85,B 0,C 180,E1 -24273.755,E2 -24273.755} C_VEL
LIN {X 0,Y 143.255,Z 256.611,A -85,B 0,C 180,E1 -24279.899,E2 -24279.899} C_VEL
LIN {X 0,Y 143.312,Z 256.619,A -85,B 0,C 180,E1 -24285.791,E2 -24285.791} C_VEL
LIN {X 0,Y 143.535,Z 256.605,A -85,B 0,C 180,E1 -24288.69,E2 -24288.69} C_VEL
LIN {X 0,Y 143.604,Z 256.585,A -85,B 0,C 180,E1 -24291.542,E2 -24291.542} C_VEL
LIN {X 0,Y 144.138,Z 256.499,A -85,B 0,C 180,E1 -24299.984,E2 -24299.984} C_VEL
LIN {X 0,Y 143.596,Z 256.584,A -85,B 0,C 180,E1 -24308.427,E2 -24308.427} C_VEL
LIN {X 0,Y 143.489,Z 256.603,A -85,B 0,C 180,E1 -24311.603,E2 -24311.603} C_VEL
LIN {X 0,Y 143.27,Z 256.625,A -85,B 0,C 180,E1 -24317.099,E2 -24317.099} C_VEL
LIN {X 0,Y 143.256,Z 256.634,A -85,B 0,C 180,E1 -24321.236,E2 -24321.236} C_VEL
LIN {X 0,Y 143.16,Z 256.618,A -85,B 0,C 180,E1 -24327.916,E2 -24327.916} C_VEL
LIN {X 0,Y 143.108,Z 256.605,A -85,B 0,C 180,E1 -24333.4,E2 -24333.4} C_VEL
LIN {X 0,Y 143.021,Z 256.67,A -85,B 0,C 180,E1 -24339.68,E2 -24339.68} C_VEL
LIN {X 0,Y 142.999,Z 256.66,A -85,B 0,C 180,E1 -24343.452,E2 -24343.452} C_VEL
LIN {X 0,Y 143.003,Z 256.672,A -85,B 0,C 180,E1 -24347.465,E2 -24347.465} C_VEL
LIN {X 0,Y 143.036,Z 256.662,A -85,B 0,C 180,E1 -24351.797,E2 -24351.797} C_VEL
LIN {X 0,Y 143.14,Z 256.649,A -85,B 0,C 180,E1 -24357.311,E2 -24357.311} C_VEL
LIN {X 0,Y 143.149,Z 256.651,A -85,B 0,C 180,E1 -24362.054,E2 -24362.054} C_VEL
LIN {X 0,Y 143.267,Z 256.642,A -85,B 0,C 180,E1 -24368.704,E2 -24368.704} C_VEL
LIN {X 0,Y 143.285,Z 256.657,A -85,B 0,C 180,E1 -24372.885,E2 -24372.885} C_VEL
LIN {X 0,Y 144.215,Z 259.336,A -85,B 0,C 180,E1 -24373.395,E2 -24373.395} C_VEL
LIN {X 0,Y 146.186,Z 261.99,A -85,B 0,C 180,E1 -24374.229,E2 -24374.229} C_VEL
LIN {X 0,Y 153.702,Z 274.048,A -85,B 0,C 180,E1 -24377.271,E2 -24377.271} C_VEL
LIN {X 0,Y 164.113,Z 293.826,A -85,B 0,C 180,E1 -24381.12,E2 -24381.12} C_VEL
LIN {X 0,Y 168.006,Z 304.002,A -85,B 0,C 180,E1 -24382.564,E2 -24382.564} C_VEL
LIN {X 0,Y 164.644,Z 354.148,A -85,B 0,C 180,E1 -24384.739,E2 -24384.739} C_VEL
LIN {X 0,Y 163.07,Z 366.878,A -85,B 0,C 180,E1 -24385.677,E2 -24385.677} C_VEL
LIN {X 0,Y 161.231,Z 379.166,A -85,B 0,C 180,E1 -24387.062,E2 -24387.062} C_VEL
LIN {X 0,Y 158.962,Z 390.322,A -85,B 0,C 180,E1 -24388.733,E2 -24388.733} C_VEL
LIN {X 0,Y 156.179,Z 401.65,A -85,B 0,C 180,E1 -24390.967,E2 -24390.967} C_VEL
LIN {X 0,Y 153.243,Z 412.071,A -85,B 0,C 180,E1 -24393.615,E2 -24393.615} C_VEL
LIN {X 0,Y 150.193,Z 421.702,A -85,B 0,C 180,E1 -24396.718,E2 -24396.718} C_VEL
LIN {X 0,Y 147.411,Z 430.366,A -85,B 0,C 180,E1 -24400.299,E2 -24400.299} C_VEL
LIN {X 0,Y 144.732,Z 438.605,A -85,B 0,C 180,E1 -24404.696,E2 -24404.696} C_VEL
LIN {X 0,Y 142.954,Z 444.346,A -85,B 0,C 180,E1 -24408.635,E2 -24408.635} C_VEL
LIN {X 0,Y 141.564,Z 449.696,A -85,B 0,C 180,E1 -24413.4,E2 -24413.4} C_VEL
LIN {X 0,Y 140.551,Z 453.695,A -85,B 0,C 180,E1 -24418.36,E2 -24418.36} C_VEL
LIN {X 0,Y 140.225,Z 456.414,A -85,B 0,C 180,E1 -24423.456,E2 -24423.456} C_VEL
LIN {X 0,Y 140.465,Z 457.547,A -85,B 0,C 180,E1 -24426.898,E2 -24426.898} C_VEL
LIN {X 0,Y 141.467,Z 458.134,A -85,B 0,C 180,E1 -24431.853,E2 -24431.853} C_VEL
LIN {X 0,Y 143.526,Z 457.405,A -85,B 0,C 180,E1 -24437.263,E2 -24437.263} C_VEL
LIN {X 0,Y 145.725,Z 455.92,A -85,B 0,C 180,E1 -24441.197,E2 -24441.197} C_VEL
LIN {X 0,Y 148.902,Z 453.216,A -85,B 0,C 180,E1 -24445.522,E2 -24445.522} C_VEL
LIN {X 0,Y 152.775,Z 449.395,A -85,B 0,C 180,E1 -24449.62,E2 -24449.62} C_VEL
LIN {X 0,Y 158.238,Z 443.404,A -85,B 0,C 180,E1 -24454.071,E2 -24454.071} C_VEL
LIN {X 0,Y 164.054,Z 436.018,A -85,B 0,C 180,E1 -24457.934,E2 -24457.934} C_VEL
LIN {X 0,Y 169.371,Z 428.408,A -85,B 0,C 180,E1 -24460.905,E2 -24460.905} C_VEL
LIN {X 0,Y 174.064,Z 420.851,A -85,B 0,C 180,E1 -24463.206,E2 -24463.206} C_VEL
LIN {X 0,Y 179.573,Z 410.677,A -85,B 0,C 180,E1 -24465.608,E2 -24465.608} C_VEL
LIN {X 0,Y 184.606,Z 399.424,A -85,B 0,C 180,E1 -24467.631,E2 -24467.631} C_VEL
LIN {X 0,Y 188.98,Z 387.68,A -85,B 0,C 180,E1 -24469.199,E2 -24469.199} C_VEL
LIN {X 0,Y 192.429,Z 375.48,A -85,B 0,C 180,E1 -24470.429,E2 -24470.429} C_VEL
LIN {X 0,Y 195.198,Z 362.254,A -85,B 0,C 180,E1 -24471.349,E2 -24471.349} C_VEL
LIN {X 0,Y 197.008,Z 348.483,A -85,B 0,C 180,E1 -24471.944,E2 -24471.944} C_VEL
LIN {X 0,Y 199.095,Z 326.106,A -85,B 0,C 180,E1 -24472.733,E2 -24472.733} C_VEL
LIN {X 0,Y 195.479,Z 318.722,A -85,B 0,C 180,E1 -24475.469,E2 -24475.469} C_VEL
LIN {X 0,Y 191.723,Z 311.664,A -85,B 0,C 180,E1 -24478.79,E2 -24478.79} C_VEL
LIN {X 0,Y 188.474,Z 306.388,A -85,B 0,C 180,E1 -24482.283,E2 -24482.283} C_VEL
LIN {X 0,Y 187.013,Z 303.646,A -85,B 0,C 180,E1 -24484.322,E2 -24484.322} C_VEL
LIN {X 0,Y 184.795,Z 301.095,A -85,B 0,C 180,E1 -24487.982,E2 -24487.982} C_VEL
LIN {X 0,Y 184.075,Z 299.107,A -85,B 0,C 180,E1 -24489.987,E2 -24489.987} C_VEL
LIN {X 0,Y 182.798,Z 298.552,A -85,B 0,C 180,E1 -24496.025,E2 -24496.025} C_VEL
LIN {X 0,Y 183.791,Z 299.337,A -85,B 0,C 180,E1 -24501.88,E2 -24501.88} C_VEL
LIN {X 0,Y 185.226,Z 302.426,A -85,B 0,C 180,E1 -24505.559,E2 -24505.559} C_VEL
LIN {X 0,Y 187.282,Z 306.206,A -85,B 0,C 180,E1 -24508.894,E2 -24508.894} C_VEL
LIN {X 0,Y 189.654,Z 311.052,A -85,B 0,C 180,E1 -24511.917,E2 -24511.917} C_VEL
LIN {X 0,Y 192.09,Z 316.368,A -85,B 0,C 180,E1 -24514.508,E2 -24514.508} C_VEL
LIN {X 0,Y 194.817,Z 322.625,A -85,B 0,C 180,E1 -24516.969,E2 -24516.969} C_VEL
LIN {X 0,Y 197.834,Z 330.695,A -85,B 0,C 180,E1 -24519.466,E2 -24519.466} C_VEL
LIN {X 0,Y 198.587,Z 333.092,A -85,B 0,C 180,E1 -24520.056,E2 -24520.056} C_VEL
LIN {X 0,Y 195.541,Z 363.632,A -85,B 0,C 180,E1 -24521.152,E2 -24521.152} C_VEL
LIN {X 0,Y 193.087,Z 376.848,A -85,B 0,C 180,E1 -24521.852,E2 -24521.852} C_VEL
LIN {X 0,Y 189.778,Z 389.263,A -85,B 0,C 180,E1 -24522.803,E2 -24522.803} C_VEL
LIN {X 0,Y 185.811,Z 400.813,A -85,B 0,C 180,E1 -24524.059,E2 -24524.059} C_VEL
LIN {X 0,Y 181.074,Z 412.033,A -85,B 0,C 180,E1 -24525.684,E2 -24525.684} C_VEL
LIN {X 0,Y 175.964,Z 422.246,A -85,B 0,C 180,E1 -24527.626,E2 -24527.626} C_VEL
LIN {X 0,Y 170.038,Z 432.351,A -85,B 0,C 180,E1 -24530.162,E2 -24530.162} C_VEL
LIN {X 0,Y 164.257,Z 441.25,A -85,B 0,C 180,E1 -24533.202,E2 -24533.202} C_VEL
LIN {X 0,Y 158.859,Z 448.494,A -85,B 0,C 180,E1 -24536.428,E2 -24536.428} C_VEL
LIN {X 0,Y 153.975,Z 454.681,A -85,B 0,C 180,E1 -24540.162,E2 -24540.162} C_VEL
LIN {X 0,Y 150.195,Z 458.991,A -85,B 0,C 180,E1 -24543.608,E2 -24543.608} C_VEL
LIN {X 0,Y 146.278,Z 463.092,A -85,B 0,C 180,E1 -24548.188,E2 -24548.188} C_VEL
LIN {X 0,Y 144.139,Z 464.6,A -85,B 0,C 180,E1 -24550.292,E2 -24550.292} C_VEL
LIN {X 0,Y 139.373,Z 466.409,A -85,B 0,C 180,E1 -24553.736,E2 -24553.736} C_VEL
LIN {X 0,Y 135.848,Z 467.254,A -85,B 0,C 180,E1 -24556.675,E2 -24556.675} C_VEL
LIN {X 0,Y 134.206,Z 467.592,A -85,B 0,C 180,E1 -24559.078,E2 -24559.078} C_VEL
LIN {X 0,Y 133.97,Z 467.626,A -85,B 0,C 180,E1 -24559.913,E2 -24559.913} C_VEL
LIN {X 0,Y 133.562,Z 467.531,A -85,B 0,C 180,E1 -24563.959,E2 -24563.959} C_VEL
LIN {X 0,Y 133.593,Z 466.456,A -85,B 0,C 180,E1 -24568.796,E2 -24568.796} C_VEL
LIN {X 0,Y 133.598,Z 464.636,A -85,B 0,C 180,E1 -24573.016,E2 -24573.016} C_VEL
LIN {X 0,Y 133.769,Z 461.676,A -85,B 0,C 180,E1 -24577.547,E2 -24577.547} C_VEL
LIN {X 0,Y 134.416,Z 457.611,A -85,B 0,C 180,E1 -24582.072,E2 -24582.072} C_VEL
LIN {X 0,Y 135.99,Z 451.302,A -85,B 0,C 180,E1 -24587.287,E2 -24587.287} C_VEL
LIN {X 0,Y 138.248,Z 444.419,A -85,B 0,C 180,E1 -24591.627,E2 -24591.627} C_VEL
LIN {X 0,Y 140.556,Z 437.352,A -85,B 0,C 180,E1 -24595.151,E2 -24595.151} C_VEL
LIN {X 0,Y 143.481,Z 428.854,A -85,B 0,C 180,E1 -24598.526,E2 -24598.526} C_VEL
LIN {X 0,Y 146.787,Z 418.313,A -85,B 0,C 180,E1 -24601.78,E2 -24601.78} C_VEL
LIN {X 0,Y 149.447,Z 409.357,A -85,B 0,C 180,E1 -24603.947,E2 -24603.947} C_VEL
LIN {X 0,Y 152.281,Z 398.341,A -85,B 0,C 180,E1 -24606.045,E2 -24606.045} C_VEL
LIN {X 0,Y 154.956,Z 386.281,A -85,B 0,C 180,E1 -24607.754,E2 -24607.754} C_VEL
LIN {X 0,Y 157.047,Z 373.471,A -85,B 0,C 180,E1 -24609.043,E2 -24609.043} C_VEL
LIN {X 0,Y 158.465,Z 360.592,A -85,B 0,C 180,E1 -24609.878,E2 -24609.878} C_VEL
LIN {X 0,Y 161.046,Z 320.888,A -85,B 0,C 180,E1 -24611.662,E2 -24611.662} C_VEL
LIN {X 0,Y 159.905,Z 309.828,A -85,B 0,C 180,E1 -24612.576,E2 -24612.576} C_VEL
LIN {X 0,Y 154.137,Z 293.582,A -85,B 0,C 180,E1 -24615.013,E2 -24615.013} C_VEL
LIN {X 0,Y 148.549,Z 280.582,A -85,B 0,C 180,E1 -24617.436,E2 -24617.436} C_VEL
LIN {X 0,Y 143.16,Z 269.569,A -85,B 0,C 180,E1 -24619.874,E2 -24619.874} C_VEL
LIN {X 0,Y 138.728,Z 262.41,A -85,B 0,C 180,E1 -24621.939,E2 -24621.939} C_VEL
LIN {X 0,Y 136.663,Z 259.667,A -85,B 0,C 180,E1 -24622.922,E2 -24622.922} C_VEL
LIN {X 0,Y 136.061,Z 257.535,A -85,B 0,C 180,E1 -24623.425,E2 -24623.425} C_VEL
LIN {X 0,Y 136.055,Z 257.534,A -85,B 0,C 180,E1 -24628.881,E2 -24628.881} C_VEL
LIN {X 0,Y 136.096,Z 257.528,A -85,B 0,C 180,E1 -24632.288,E2 -24632.288} C_VEL
LIN {X 0,Y 136.19,Z 257.503,A -85,B 0,C 180,E1 -24638.808,E2 -24638.808} C_VEL
LIN {X 0,Y 136.231,Z 257.49,A -85,B 0,C 180,E1 -24645.035,E2 -24645.035} C_VEL
LIN {X 0,Y 136.43,Z 257.49,A -85,B 0,C 180,E1 -24648.163,E2 -24648.163} C_VEL
LIN {X 0,Y 136.535,Z 257.468,A -85,B 0,C 180,E1 -24651.1,E2 -24651.1} C_VEL
LIN {X 0,Y 137.094,Z 257.373,A -85,B 0,C 180,E1 -24659.983,E2 -24659.983} C_VEL
LIN {X 0,Y 136.525,Z 257.462,A -85,B 0,C 180,E1 -24668.866,E2 -24668.866} C_VEL
LIN {X 0,Y 136.405,Z 257.487,A -85,B 0,C 180,E1 -24671.876,E2 -24671.876} C_VEL
LIN {X 0,Y 136.187,Z 257.502,A -85,B 0,C 180,E1 -24678.018,E2 -24678.018} C_VEL
LIN {X 0,Y 136.177,Z 257.518,A -85,B 0,C 180,E1 -24681.729,E2 -24681.729} C_VEL
LIN {X 0,Y 136.069,Z 257.491,A -85,B 0,C 180,E1 -24688.594,E2 -24688.594} C_VEL
LIN {X 0,Y 136.011,Z 257.502,A -85,B 0,C 180,E1 -24694.616,E2 -24694.616} C_VEL
LIN {X 0,Y 135.993,Z 257.544,A -85,B 0,C 180,E1 -24699.18,E2 -24699.18} C_VEL
LIN {X 0,Y 135.944,Z 257.538,A -85,B 0,C 180,E1 -24703.635,E2 -24703.635} C_VEL
LIN {X 0,Y 135.947,Z 257.55,A -85,B 0,C 180,E1 -24707.775,E2 -24707.775} C_VEL
LIN {X 0,Y 135.985,Z 257.539,A -85,B 0,C 180,E1 -24711.671,E2 -24711.671} C_VEL
LIN {X 0,Y 136.015,Z 257.538,A -85,B 0,C 180,E1 -24715.73,E2 -24715.73} C_VEL
LIN {X 0,Y 136.105,Z 257.528,A -85,B 0,C 180,E1 -24722.308,E2 -24722.308} C_VEL
LIN {X 0,Y 136.265,Z 257.52,A -85,B 0,C 180,E1 -24730.022,E2 -24730.022} C_VEL
LIN {X 0,Y 136.249,Z 257.532,A -85,B 0,C 180,E1 -24730.412,E2 -24730.412} C_VEL
LIN {X 0,Y 137.225,Z 260.333,A -85,B 0,C 180,E1 -24730.998,E2 -24730.998} C_VEL
LIN {X 0,Y 139.071,Z 262.69,A -85,B 0,C 180,E1 -24731.86,E2 -24731.86} C_VEL
LIN {X 0,Y 141.295,Z 266.124,A -85,B 0,C 180,E1 -24732.906,E2 -24732.906} C_VEL
LIN {X 0,Y 149.514,Z 279.476,A -85,B 0,C 180,E1 -24736.445,E2 -24736.445} C_VEL
LIN {X 0,Y 158.826,Z 297.599,A -85,B 0,C 180,E1 -24740.096,E2 -24740.096} C_VEL
LIN {X 0,Y 161.941,Z 306.018,A -85,B 0,C 180,E1 -24741.336,E2 -24741.336} C_VEL
LIN {X 0,Y 158.438,Z 354.772,A -85,B 0,C 180,E1 -24743.505,E2 -24743.505} C_VEL
LIN {X 0,Y 156.791,Z 367.882,A -85,B 0,C 180,E1 -24744.529,E2 -24744.529} C_VEL
LIN {X 0,Y 154.673,Z 380.819,A -85,B 0,C 180,E1 -24746.062,E2 -24746.062} C_VEL
LIN {X 0,Y 152.03,Z 392.801,A -85,B 0,C 180,E1 -24748.013,E2 -24748.013} C_VEL
LIN {X 0,Y 148.952,Z 404.52,A -85,B 0,C 180,E1 -24750.536,E2 -24750.536} C_VEL
LIN {X 0,Y 145.791,Z 414.946,A -85,B 0,C 180,E1 -24753.454,E2 -24753.454} C_VEL
LIN {X 0,Y 142.505,Z 424.646,A -85,B 0,C 180,E1 -24756.95,E2 -24756.95} C_VEL
LIN {X 0,Y 139.705,Z 433.103,A -85,B 0,C 180,E1 -24760.873,E2 -24760.873} C_VEL
LIN {X 0,Y 137.421,Z 439.799,A -85,B 0,C 180,E1 -24764.815,E2 -24764.815} C_VEL
LIN {X 0,Y 135.562,Z 445.797,A -85,B 0,C 180,E1 -24769.351,E2 -24769.351} C_VEL
LIN {X 0,Y 134.145,Z 451.165,A -85,B 0,C 180,E1 -24774.779,E2 -24774.779} C_VEL
LIN {X 0,Y 133.245,Z 454.867,A -85,B 0,C 180,E1 -24780.07,E2 -24780.07} C_VEL
LIN {X 0,Y 133.204,Z 457.232,A -85,B 0,C 180,E1 -24785.475,E2 -24785.475} C_VEL
LIN {X 0,Y 133.686,Z 458.097,A -85,B 0,C 180,E1 -24789.111,E2 -24789.111} C_VEL
LIN {X 0,Y 134.691,Z 458.401,A -85,B 0,C 180,E1 -24793.1,E2 -24793.1} C_VEL
LIN {X 0,Y 136.705,Z 457.786,A -85,B 0,C 180,E1 -24798.087,E2 -24798.087} C_VEL
LIN {X 0,Y 139.925,Z 455.778,A -85,B 0,C 180,E1 -24803.476,E2 -24803.476} C_VEL
LIN {X 0,Y 144.256,Z 452.261,A -85,B 0,C 180,E1 -24808.641,E2 -24808.641} C_VEL
LIN {X 0,Y 149.449,Z 447.282,A -85,B 0,C 180,E1 -24813.312,E2 -24813.312} C_VEL
LIN {X 0,Y 154.58,Z 441.727,A -85,B 0,C 180,E1 -24817.02,E2 -24817.02} C_VEL
LIN {X 0,Y 160.307,Z 434.74,A -85,B 0,C 180,E1 -24820.48,E2 -24820.48} C_VEL
LIN {X 0,Y 165.86,Z 427.015,A -85,B 0,C 180,E1 -24823.341,E2 -24823.341} C_VEL
LIN {X 0,Y 171.857,Z 417.397,A -85,B 0,C 180,E1 -24826.041,E2 -24826.041} C_VEL
LIN {X 0,Y 177.59,Z 406.49,A -85,B 0,C 180,E1 -24828.36,E2 -24828.36} C_VEL
LIN {X 0,Y 182.739,Z 394.574,A -85,B 0,C 180,E1 -24830.227,E2 -24830.227} C_VEL
LIN {X 0,Y 186.983,Z 382.403,A -85,B 0,C 180,E1 -24831.647,E2 -24831.647} C_VEL
LIN {X 0,Y 190.236,Z 369.876,A -85,B 0,C 180,E1 -24832.712,E2 -24832.712} C_VEL
LIN {X 0,Y 192.559,Z 357.303,A -85,B 0,C 180,E1 -24833.432,E2 -24833.432} C_VEL
LIN {X 0,Y 195.461,Z 329.707,A -85,B 0,C 180,E1 -24834.439,E2 -24834.439} C_VEL
LIN {X 0,Y 192.401,Z 323.252,A -85,B 0,C 180,E1 -24836.991,E2 -24836.991} C_VEL
LIN {X 0,Y 189.64,Z 317.798,A -85,B 0,C 180,E1 -24839.705,E2 -24839.705} C_VEL
LIN {X 0,Y 186.851,Z 312.905,A -85,B 0,C 180,E1 -24842.964,E2 -24842.964} C_VEL
LIN {X 0,Y 185.537,Z 310.415,A -85,B 0,C 180,E1 -24844.901,E2 -24844.901} C_VEL
LIN {X 0,Y 183.459,Z 307.69,A -85,B 0,C 180,E1 -24848.687,E2 -24848.687} C_VEL
LIN {X 0,Y 182.932,Z 306.057,A -85,B 0,C 180,E1 -24850.309,E2 -24850.309} C_VEL
LIN {X 0,Y 181.808,Z 305.585,A -85,B 0,C 180,E1 -24855.712,E2 -24855.712} C_VEL
LIN {X 0,Y 182.678,Z 306.294,A -85,B 0,C 180,E1 -24861.597,E2 -24861.597} C_VEL
LIN {X 0,Y 184.321,Z 310.116,A -85,B 0,C 180,E1 -24865.887,E2 -24865.887} C_VEL
LIN {X 0,Y 185.668,Z 312.628,A -85,B 0,C 180,E1 -24868.122,E2 -24868.122} C_VEL
LIN {X 0,Y 187.866,Z 317.54,A -85,B 0,C 180,E1 -24871.2,E2 -24871.2} C_VEL
LIN {X 0,Y 190.365,Z 323.352,A -85,B 0,C 180,E1 -24874.012,E2 -24874.012} C_VEL
LIN {X 0,Y 193.34,Z 331.021,A -85,B 0,C 180,E1 -24876.87,E2 -24876.87} C_VEL
LIN {X 0,Y 194.978,Z 335.922,A -85,B 0,C 180,E1 -24878.327,E2 -24878.327} C_VEL
LIN {X 0,Y 191.996,Z 363.836,A -85,B 0,C 180,E1 -24879.329,E2 -24879.329} C_VEL
LIN {X 0,Y 189.363,Z 377.283,A -85,B 0,C 180,E1 -24880.046,E2 -24880.046} C_VEL
LIN {X 0,Y 186.078,Z 389.036,A -85,B 0,C 180,E1 -24880.943,E2 -24880.943} C_VEL
LIN {X 0,Y 182.264,Z 399.815,A -85,B 0,C 180,E1 -24882.077,E2 -24882.077} C_VEL
LIN {X 0,Y 177.353,Z 411.161,A -85,B 0,C 180,E1 -24883.683,E2 -24883.683} C_VEL
LIN {X 0,Y 171.999,Z 421.483,A -85,B 0,C 180,E1 -24885.596,E2 -24885.596} C_VEL
LIN {X 0,Y 165.805,Z 431.7,A -85,B 0,C 180,E1 -24888.12,E2 -24888.12} C_VEL
LIN {X 0,Y 160.657,Z 439.288,A -85,B 0,C 180,E1 -24890.633,E2 -24890.633} C_VEL
LIN {X 0,Y 154.84,Z 446.791,A -85,B 0,C 180,E1 -24893.84,E2 -24893.84} C_VEL
LIN {X 0,Y 149.692,Z 452.886,A -85,B 0,C 180,E1 -24897.323,E2 -24897.323} C_VEL
LIN {X 0,Y 145.276,Z 457.783,A -85,B 0,C 180,E1 -24901.069,E2 -24901.069} C_VEL
LIN {X 0,Y 141.379,Z 461.612,A -85,B 0,C 180,E1 -24905.006,E2 -24905.006} C_VEL
LIN {X 0,Y 138.213,Z 464.464,A -85,B 0,C 180,E1 -24909.149,E2 -24909.149} C_VEL
LIN {X 0,Y 136.51,Z 465.844,A -85,B 0,C 180,E1 -24912.008,E2 -24912.008} C_VEL
LIN {X 0,Y 134.385,Z 467.478,A -85,B 0,C 180,E1 -24917.926,E2 -24917.926} C_VEL
LIN {X 0,Y 133.97,Z 467.626,A -85,B 0,C 180,E1 -24919.913,E2 -24919.913} C_VEL
LIN {X 0,Y 133.006,Z 467.646,A -85,B 0,C 180,E1 -24922.419,E2 -24922.419} C_VEL
LIN {X 0,Y 131.319,Z 467.344,A -85,B 0,C 180,E1 -24924.891,E2 -24924.891} C_VEL
LIN {X 0,Y 127.652,Z 465.765,A -85,B 0,C 180,E1 -24929.912,E2 -24929.912} C_VEL
LIN {X 0,Y 126.517,Z 463.956,A -85,B 0,C 180,E1 -24933.392,E2 -24933.392} C_VEL
LIN {X 0,Y 126.71,Z 461.007,A -85,B 0,C 180,E1 -24937.971,E2 -24937.971} C_VEL
LIN {X 0,Y 127.437,Z 456.816,A -85,B 0,C 180,E1 -24942.744,E2 -24942.744} C_VEL
LIN {X 0,Y 129.2,Z 450.375,A -85,B 0,C 180,E1 -24948.227,E2 -24948.227} C_VEL
LIN {X 0,Y 131.603,Z 443.324,A -85,B 0,C 180,E1 -24952.778,E2 -24952.778} C_VEL
LIN {X 0,Y 134.432,Z 435.102,A -85,B 0,C 180,E1 -24956.88,E2 -24956.88} C_VEL
LIN {X 0,Y 137.216,Z 427.315,A -85,B 0,C 180,E1 -24959.957,E2 -24959.957} C_VEL
LIN {X 0,Y 140.369,Z 417.685,A -85,B 0,C 180,E1 -24962.989,E2 -24962.989} C_VEL
LIN {X 0,Y 143.167,Z 408.657,A -85,B 0,C 180,E1 -24965.225,E2 -24965.225} C_VEL
LIN {X 0,Y 146.125,Z 397.538,A -85,B 0,C 180,E1 -24967.387,E2 -24967.387} C_VEL
LIN {X 0,Y 148.894,Z 385.295,A -85,B 0,C 180,E1 -24969.146,E2 -24969.146} C_VEL
LIN {X 0,Y 151.16,Z 371.651,A -85,B 0,C 180,E1 -24970.5,E2 -24970.5} C_VEL
LIN {X 0,Y 152.549,Z 358.657,A -85,B 0,C 180,E1 -24971.319,E2 -24971.319} C_VEL
LIN {X 0,Y 155.029,Z 321.652,A -85,B 0,C 180,E1 -24973.021,E2 -24973.021} C_VEL
LIN {X 0,Y 154.117,Z 312.168,A -85,B 0,C 180,E1 -24973.839,E2 -24973.839} C_VEL
LIN {X 0,Y 148.504,Z 296.195,A -85,B 0,C 180,E1 -24976.398,E2 -24976.398} C_VEL
LIN {X 0,Y 143.476,Z 284.347,A -85,B 0,C 180,E1 -24978.711,E2 -24978.711} C_VEL
LIN {X 0,Y 138.682,Z 274.299,A -85,B 0,C 180,E1 -24981.054,E2 -24981.054} C_VEL
LIN {X 0,Y 133.598,Z 266.357,A -85,B 0,C 180,E1 -24983.579,E2 -24983.579} C_VEL
LIN {X 0,Y 131.41,Z 262.892,A -85,B 0,C 180,E1 -24984.743,E2 -24984.743} C_VEL
LIN {X 0,Y 129.712,Z 260.713,A -85,B 0,C 180,E1 -24985.646,E2 -24985.646} C_VEL
LIN {X 0,Y 129.016,Z 258.419,A -85,B 0,C 180,E1 -24986.208,E2 -24986.208} C_VEL
LIN {X 0,Y 128.994,Z 258.42,A -85,B 0,C 180,E1 -24990.658,E2 -24990.658} C_VEL
LIN {X 0,Y 129.078,Z 258.4,A -85,B 0,C 180,E1 -24997.758,E2 -24997.758} C_VEL
LIN {X 0,Y 129.153,Z 258.36,A -85,B 0,C 180,E1 -25004.195,E2 -25004.195} C_VEL
LIN {X 0,Y 129.348,Z 258.372,A -85,B 0,C 180,E1 -25007.956,E2 -25007.956} C_VEL
LIN {X 0,Y 129.462,Z 258.352,A -85,B 0,C 180,E1 -25010.61,E2 -25010.61} C_VEL
LIN {X 0,Y 130.049,Z 258.247,A -85,B 0,C 180,E1 -25019.982,E2 -25019.982} C_VEL
LIN {X 0,Y 129.451,Z 258.342,A -85,B 0,C 180,E1 -25029.355,E2 -25029.355} C_VEL
LIN {X 0,Y 129.289,Z 258.377,A -85,B 0,C 180,E1 -25032.54,E2 -25032.54} C_VEL
LIN {X 0,Y 129.11,Z 258.383,A -85,B 0,C 180,E1 -25039.043,E2 -25039.043} C_VEL
LIN {X 0,Y 129.089,Z 258.402,A -85,B 0,C 180,E1 -25042.381,E2 -25042.381} C_VEL
LIN {X 0,Y 128.993,Z 258.36,A -85,B 0,C 180,E1 -25049.341,E2 -25049.341} C_VEL
LIN {X 0,Y 128.927,Z 258.388,A -85,B 0,C 180,E1 -25055.149,E2 -25055.149} C_VEL
LIN {X 0,Y 128.89,Z 258.428,A -85,B 0,C 180,E1 -25060.842,E2 -25060.842} C_VEL
LIN {X 0,Y 128.878,Z 258.425,A -85,B 0,C 180,E1 -25065.119,E2 -25065.119} C_VEL
LIN {X 0,Y 128.898,Z 258.418,A -85,B 0,C 180,E1 -25069.727,E2 -25069.727} C_VEL
LIN {X 0,Y 128.919,Z 258.426,A -85,B 0,C 180,E1 -25074.822,E2 -25074.822} C_VEL
LIN {X 0,Y 128.976,Z 258.423,A -85,B 0,C 180,E1 -25080.633,E2 -25080.633} C_VEL
LIN {X 0,Y 129.103,Z 258.403,A -85,B 0,C 180,E1 -25087.548,E2 -25087.548} C_VEL
LIN {X 0,Y 130.043,Z 261.068,A -85,B 0,C 180,E1 -25088.205,E2 -25088.205} C_VEL
LIN {X 0,Y 132.225,Z 263.78,A -85,B 0,C 180,E1 -25089.345,E2 -25089.345} C_VEL
LIN {X 0,Y 134.459,Z 267.17,A -85,B 0,C 180,E1 -25090.503,E2 -25090.503} C_VEL
LIN {X 0,Y 142.841,Z 280.568,A -85,B 0,C 180,E1 -25094.485,E2 -25094.485} C_VEL
LIN {X 0,Y 148.797,Z 291.889,A -85,B 0,C 180,E1 -25097.072,E2 -25097.072} C_VEL
LIN {X 0,Y 153.909,Z 302.138,A -85,B 0,C 180,E1 -25099.136,E2 -25099.136} C_VEL
LIN {X 0,Y 155.897,Z 307.527,A -85,B 0,C 180,E1 -25099.983,E2 -25099.983} C_VEL
LIN {X 0,Y 152.4,Z 354.638,A -85,B 0,C 180,E1 -25102.131,E2 -25102.131} C_VEL
LIN {X 0,Y 150.732,Z 367.46,A -85,B 0,C 180,E1 -25103.138,E2 -25103.138} C_VEL
LIN {X 0,Y 148.752,Z 379.523,A -85,B 0,C 180,E1 -25104.578,E2 -25104.578} C_VEL
LIN {X 0,Y 145.941,Z 392.082,A -85,B 0,C 180,E1 -25106.61,E2 -25106.61} C_VEL
LIN {X 0,Y 142.588,Z 404.325,A -85,B 0,C 180,E1 -25109.294,E2 -25109.294} C_VEL
LIN {X 0,Y 139.244,Z 414.95,A -85,B 0,C 180,E1 -25112.349,E2 -25112.349} C_VEL
LIN {X 0,Y 135.873,Z 424.565,A -85,B 0,C 180,E1 -25115.938,E2 -25115.938} C_VEL
LIN {X 0,Y 132.981,Z 432.811,A -85,B 0,C 180,E1 -25119.89,E2 -25119.89} C_VEL
LIN {X 0,Y 130.465,Z 439.939,A -85,B 0,C 180,E1 -25124.24,E2 -25124.24} C_VEL
LIN {X 0,Y 128.46,Z 446.128,A -85,B 0,C 180,E1 -25129.162,E2 -25129.162} C_VEL
LIN {X 0,Y 127.085,Z 451.169,A -85,B 0,C 180,E1 -25134.503,E2 -25134.503} C_VEL
LIN {X 0,Y 126.152,Z 454.937,A -85,B 0,C 180,E1 -25140.091,E2 -25140.091} C_VEL
LIN {X 0,Y 126.024,Z 456.711,A -85,B 0,C 180,E1 -25143.894,E2 -25143.894} C_VEL
LIN {X 0,Y 126.554,Z 458.199,A -85,B 0,C 180,E1 -25149.003,E2 -25149.003} C_VEL
LIN {X 0,Y 128.311,Z 458.645,A -85,B 0,C 180,E1 -25155.4,E2 -25155.4} C_VEL
LIN {X 0,Y 130.275,Z 458.008,A -85,B 0,C 180,E1 -25159.682,E2 -25159.682} C_VEL
LIN {X 0,Y 133.336,Z 456.279,A -85,B 0,C 180,E1 -25164.587,E2 -25164.587} C_VEL
LIN {X 0,Y 137.99,Z 452.905,A -85,B 0,C 180,E1 -25169.975,E2 -25169.975} C_VEL
LIN {X 0,Y 143.624,Z 447.97,A -85,B 0,C 180,E1 -25174.874,E2 -25174.874} C_VEL
LIN {X 0,Y 148.59,Z 442.992,A -85,B 0,C 180,E1 -25178.389,E2 -25178.389} C_VEL
LIN {X 0,Y 155.032,Z 435.691,A -85,B 0,C 180,E1 -25182.167,E2 -25182.167} C_VEL
LIN {X 0,Y 161.594,Z 427.082,A -85,B 0,C 180,E1 -25185.39,E2 -25185.39} C_VEL
LIN {X 0,Y 167.884,Z 417.433,A -85,B 0,C 180,E1 -25188.088,E2 -25188.088} C_VEL
LIN {X 0,Y 173.271,Z 407.744,A -85,B 0,C 180,E1 -25190.154,E2 -25190.154} C_VEL
LIN {X 0,Y 178.35,Z 396.835,A -85,B 0,C 180,E1 -25191.906,E2 -25191.906} C_VEL
LIN {X 0,Y 182.975,Z 384.456,A -85,B 0,C 180,E1 -25193.396,E2 -25193.396} C_VEL
LIN {X 0,Y 186.493,Z 372.182,A -85,B 0,C 180,E1 -25194.473,E2 -25194.473} C_VEL
LIN {X 0,Y 188.911,Z 360.332,A -85,B 0,C 180,E1 -25195.199,E2 -25195.199} C_VEL
LIN {X 0,Y 190.841,Z 345.024,A -85,B 0,C 180,E1 -25195.788,E2 -25195.788} C_VEL
LIN {X 0,Y 192.048,Z 333.327,A -85,B 0,C 180,E1 -25196.188,E2 -25196.188} C_VEL
LIN {X 0,Y 188.667,Z 325.967,A -85,B 0,C 180,E1 -25199.485,E2 -25199.485} C_VEL
LIN {X 0,Y 185.546,Z 319.966,A -85,B 0,C 180,E1 -25203.245,E2 -25203.245} C_VEL
LIN {X 0,Y 184.155,Z 317.229,A -85,B 0,C 180,E1 -25205.382,E2 -25205.382} C_VEL
LIN {X 0,Y 182.122,Z 314.24,A -85,B 0,C 180,E1 -25209.475,E2 -25209.475} C_VEL
LIN {X 0,Y 181.785,Z 313.08,A -85,B 0,C 180,E1 -25210.636,E2 -25210.636} C_VEL
LIN {X 0,Y 180.796,Z 312.616,A -85,B 0,C 180,E1 -25215.802,E2 -25215.802} C_VEL
LIN {X 0,Y 181.596,Z 313.329,A -85,B 0,C 180,E1 -25221.417,E2 -25221.417} C_VEL
LIN {X 0,Y 183.059,Z 317.039,A -85,B 0,C 180,E1 -25225.493,E2 -25225.493} C_VEL
LIN {X 0,Y 184.228,Z 319.473,A -85,B 0,C 180,E1 -25227.592,E2 -25227.592} C_VEL
LIN {X 0,Y 186.128,Z 324.104,A -85,B 0,C 180,E1 -25230.498,E2 -25230.498} C_VEL
LIN {X 0,Y 188.385,Z 329.689,A -85,B 0,C 180,E1 -25233.211,E2 -25233.211} C_VEL
LIN {X 0,Y 191.075,Z 337.455,A -85,B 0,C 180,E1 -25236.063,E2 -25236.063} C_VEL
LIN {X 0,Y 191.54,Z 339.01,A -85,B 0,C 180,E1 -25236.523,E2 -25236.523} C_VEL
LIN {X 0,Y 188.698,Z 364.279,A -85,B 0,C 180,E1 -25237.442,E2 -25237.442} C_VEL
LIN {X 0,Y 186.023,Z 377.341,A -85,B 0,C 180,E1 -25238.135,E2 -25238.135} C_VEL
LIN {X 0,Y 182.222,Z 390.155,A -85,B 0,C 180,E1 -25239.117,E2 -25239.117} C_VEL
LIN {X 0,Y 177.689,Z 402.027,A -85,B 0,C 180,E1 -25240.416,E2 -25240.416} C_VEL
LIN {X 0,Y 172.595,Z 412.896,A -85,B 0,C 180,E1 -25242.003,E2 -25242.003} C_VEL
LIN {X 0,Y 167.671,Z 421.789,A -85,B 0,C 180,E1 -25243.696,E2 -25243.696} C_VEL
LIN {X 0,Y 161.801,Z 431.045,A -85,B 0,C 180,E1 -25245.976,E2 -25245.976} C_VEL
LIN {X 0,Y 156.285,Z 438.711,A -85,B 0,C 180,E1 -25248.45,E2 -25248.45} C_VEL
LIN {X 0,Y 150.166,Z 446.264,A -85,B 0,C 180,E1 -25251.676,E2 -25251.676} C_VEL
LIN {X 0,Y 143.772,Z 453.303,A -85,B 0,C 180,E1 -25255.796,E2 -25255.796} C_VEL
LIN {X 0,Y 139.111,Z 458.033,A -85,B 0,C 180,E1 -25259.656,E2 -25259.656} C_VEL
LIN {X 0,Y 134.949,Z 461.722,A -85,B 0,C 180,E1 -25263.726,E2 -25263.726} C_VEL
LIN {X 0,Y 131.583,Z 464.454,A -85,B 0,C 180,E1 -25268.046,E2 -25268.046} C_VEL
LIN {X 0,Y 129.747,Z 465.777,A -85,B 0,C 180,E1 -25271.035,E2 -25271.035} C_VEL
LIN {X 0,Y 128.434,Z 466.723,A -85,B 0,C 180,E1 -25274.122,E2 -25274.122} C_VEL
LIN {X 0,Y 126.79,Z 467.408,A -85,B 0,C 180,E1 -25280.428,E2 -25280.428} C_VEL
LIN {X 0,Y 126.468,Z 466.584,A -85,B 0,C 180,E1 -25286.815,E2 -25286.815} C_VEL
LIN {X 0,Y 126.557,Z 465.119,A -85,B 0,C 180,E1 -25291.039,E2 -25291.039} C_VEL
LIN {X 0,Y 126.517,Z 463.956,A -85,B 0,C 180,E1 -25293.392,E2 -25293.392} C_VEL
LIN {X 0,Y 125.851,Z 462.41,A -85,B 0,C 180,E1 -25295.942,E2 -25295.942} C_VEL
LIN {X 0,Y 123.364,Z 459.185,A -85,B 0,C 180,E1 -25300.096,E2 -25300.096} C_VEL
LIN {X 0,Y 121.342,Z 455.221,A -85,B 0,C 180,E1 -25304.295,E2 -25304.295} C_VEL
LIN {X 0,Y 121.441,Z 452.481,A -85,B 0,C 180,E1 -25306.811,E2 -25306.811} C_VEL
LIN {X 0,Y 123.714,Z 446.009,A -85,B 0,C 180,E1 -25311.669,E2 -25311.669} C_VEL
LIN {X 0,Y 126.649,Z 437.881,A -85,B 0,C 180,E1 -25316.355,E2 -25316.355} C_VEL
LIN {X 0,Y 130.036,Z 428.78,A -85,B 0,C 180,E1 -25320.396,E2 -25320.396} C_VEL
LIN {X 0,Y 133.301,Z 419.436,A -85,B 0,C 180,E1 -25323.613,E2 -25323.613} C_VEL
LIN {X 0,Y 136.035,Z 410.752,A -85,B 0,C 180,E1 -25325.991,E2 -25325.991} C_VEL
LIN {X 0,Y 139.14,Z 400.248,A -85,B 0,C 180,E1 -25328.224,E2 -25328.224} C_VEL
LIN {X 0,Y 142.264,Z 387.742,A -85,B 0,C 180,E1 -25330.187,E2 -25330.187} C_VEL
LIN {X 0,Y 144.667,Z 374.635,A -85,B 0,C 180,E1 -25331.677,E2 -25331.677} C_VEL
LIN {X 0,Y 146.361,Z 361.158,A -85,B 0,C 180,E1 -25332.635,E2 -25332.635} C_VEL
LIN {X 0,Y 149.112,Z 322.021,A -85,B 0,C 180,E1 -25334.513,E2 -25334.513} C_VEL
LIN {X 0,Y 148.402,Z 314.48,A -85,B 0,C 180,E1 -25335.205,E2 -25335.205} C_VEL
LIN {X 0,Y 143.031,Z 299.11,A -85,B 0,C 180,E1 -25337.798,E2 -25337.798} C_VEL
LIN {X 0,Y 138.285,Z 287.679,A -85,B 0,C 180,E1 -25340.177,E2 -25340.177} C_VEL
LIN {X 0,Y 134.071,Z 278.713,A -85,B 0,C 180,E1 -25342.399,E2 -25342.399} C_VEL
LIN {X 0,Y 129.014,Z 270.724,A -85,B 0,C 180,E1 -25345.074,E2 -25345.074} C_VEL
LIN {X 0,Y 127.233,Z 267.99,A -85,B 0,C 180,E1 -25346.091,E2 -25346.091} C_VEL
LIN {X 0,Y 125.161,Z 264.64,A -85,B 0,C 180,E1 -25347.337,E2 -25347.337} C_VEL
LIN {X 0,Y 122.809,Z 262.006,A -85,B 0,C 180,E1 -25348.717,E2 -25348.717} C_VEL
LIN {X 0,Y 121.915,Z 259.298,A -85,B 0,C 180,E1 -25349.514,E2 -25349.514} C_VEL
LIN {X 0,Y 121.989,Z 259.286,A -85,B 0,C 180,E1 -25357.185,E2 -25357.185} C_VEL
LIN {X 0,Y 122.066,Z 259.234,A -85,B 0,C 180,E1 -25363.251,E2 -25363.251} C_VEL
LIN {X 0,Y 122.291,Z 259.249,A -85,B 0,C 180,E1 -25367.676,E2 -25367.676} C_VEL
LIN {X 0,Y 122.391,Z 259.236,A -85,B 0,C 180,E1 -25370.062,E2 -25370.062} C_VEL
LIN {X 0,Y 122.523,Z 259.154,A -85,B 0,C 180,E1 -25376.693,E2 -25376.693} C_VEL
LIN {X 0,Y 123.002,Z 259.121,A -85,B 0,C 180,E1 -25379.981,E2 -25379.981} C_VEL
LIN {X 0,Y 122.38,Z 259.234,A -85,B 0,C 180,E1 -25386.823,E2 -25386.823} C_VEL
LIN {X 0,Y 122.277,Z 259.248,A -85,B 0,C 180,E1 -25392.292,E2 -25392.292} C_VEL
LIN {X 0,Y 122.07,Z 259.266,A -85,B 0,C 180,E1 -25396.71,E2 -25396.71} C_VEL
LIN {X 0,Y 122.008,Z 259.285,A -85,B 0,C 180,E1 -25402.836,E2 -25402.836} C_VEL
LIN {X 0,Y 121.914,Z 259.264,A -85,B 0,C 180,E1 -25407.44,E2 -25407.44} C_VEL
LIN {X 0,Y 121.872,Z 259.233,A -85,B 0,C 180,E1 -25411.241,E2 -25411.241} C_VEL
LIN {X 0,Y 121.851,Z 259.282,A -85,B 0,C 180,E1 -25416.151,E2 -25416.151} C_VEL
LIN {X 0,Y 121.831,Z 259.304,A -85,B 0,C 180,E1 -25421.418,E2 -25421.418} C_VEL
LIN {X 0,Y 121.828,Z 259.305,A -85,B 0,C 180,E1 -25428.553,E2 -25428.553} C_VEL
LIN {X 0,Y 121.871,Z 259.304,A -85,B 0,C 180,E1 -25434.784,E2 -25434.784} C_VEL
LIN {X 0,Y 121.886,Z 259.308,A -85,B 0,C 180,E1 -25439.829,E2 -25439.829} C_VEL
LIN {X 0,Y 121.968,Z 259.296,A -85,B 0,C 180,E1 -25444.222,E2 -25444.222} C_VEL
LIN {X 0,Y 122.856,Z 261.959,A -85,B 0,C 180,E1 -25444.959,E2 -25444.959} C_VEL
LIN {X 0,Y 124.921,Z 264.214,A -85,B 0,C 180,E1 -25446.166,E2 -25446.166} C_VEL
LIN {X 0,Y 127.666,Z 268.247,A -85,B 0,C 180,E1 -25447.798,E2 -25447.798} C_VEL
LIN {X 0,Y 135.153,Z 279.922,A -85,B 0,C 180,E1 -25451.777,E2 -25451.777} C_VEL
LIN {X 0,Y 140.363,Z 288.983,A -85,B 0,C 180,E1 -25454.288,E2 -25454.288} C_VEL
LIN {X 0,Y 148.47,Z 305.299,A -85,B 0,C 180,E1 -25457.875,E2 -25457.875} C_VEL
LIN {X 0,Y 149.864,Z 308.895,A -85,B 0,C 180,E1 -25458.489,E2 -25458.489} C_VEL
LIN {X 0,Y 146.312,Z 355.886,A -85,B 0,C 180,E1 -25460.746,E2 -25460.746} C_VEL
LIN {X 0,Y 144.607,Z 368.422,A -85,B 0,C 180,E1 -25461.792,E2 -25461.792} C_VEL
LIN {X 0,Y 142.239,Z 381.526,A -85,B 0,C 180,E1 -25463.439,E2 -25463.439} C_VEL
LIN {X 0,Y 139.169,Z 394.162,A -85,B 0,C 180,E1 -25465.656,E2 -25465.656} C_VEL
LIN {X 0,Y 136.069,Z 404.9,A -85,B 0,C 180,E1 -25468.15,E2 -25468.15} C_VEL
LIN {X 0,Y 132.681,Z 415.181,A -85,B 0,C 180,E1 -25471.237,E2 -25471.237} C_VEL
LIN {X 0,Y 129.39,Z 424.11,A -85,B 0,C 180,E1 -25474.673,E2 -25474.673} C_VEL
LIN {X 0,Y 126.204,Z 432.75,A -85,B 0,C 180,E1 -25478.959,E2 -25478.959} C_VEL
LIN {X 0,Y 123.74,Z 439.358,A -85,B 0,C 180,E1 -25483.131,E2 -25483.131} C_VEL
LIN {X 0,Y 121.506,Z 446.009,A -85,B 0,C 180,E1 -25488.549,E2 -25488.549} C_VEL
LIN {X 0,Y 120.014,Z 451.137,A -85,B 0,C 180,E1 -25494.199,E2 -25494.199} C_VEL
LIN {X 0,Y 119.065,Z 454.989,A -85,B 0,C 180,E1 -25500.113,E2 -25500.113} C_VEL
LIN {X 0,Y 119.051,Z 457.555,A -85,B 0,C 180,E1 -25506.179,E2 -25506.179} C_VEL
LIN {X 0,Y 119.672,Z 458.525,A -85,B 0,C 180,E1 -25510.264,E2 -25510.264} C_VEL
LIN {X 0,Y 121.351,Z 458.942,A -85,B 0,C 180,E1 -25516.004,E2 -25516.004} C_VEL
LIN {X 0,Y 124.422,Z 458.05,A -85,B 0,C 180,E1 -25522.257,E2 -25522.257} C_VEL
LIN {X 0,Y 127.362,Z 456.475,A -85,B 0,C 180,E1 -25526.532,E2 -25526.532} C_VEL
LIN {X 0,Y 131.678,Z 453.621,A -85,B 0,C 180,E1 -25531.313,E2 -25531.313} C_VEL
LIN {X 0,Y 136.78,Z 449.612,A -85,B 0,C 180,E1 -25535.749,E2 -25535.749} C_VEL
LIN {X 0,Y 142.658,Z 444.294,A -85,B 0,C 180,E1 -25539.845,E2 -25539.845} C_VEL
LIN {X 0,Y 149.195,Z 437.462,A -85,B 0,C 180,E1 -25543.599,E2 -25543.599} C_VEL
LIN {X 0,Y 155.058,Z 430.47,A -85,B 0,C 180,E1 -25546.466,E2 -25546.466} C_VEL
LIN {X 0,Y 161.788,Z 421.261,A -85,B 0,C 180,E1 -25549.287,E2 -25549.287} C_VEL
LIN {X 0,Y 167.847,Z 411.394,A -85,B 0,C 180,E1 -25551.565,E2 -25551.565} C_VEL
LIN {X 0,Y 173.187,Z 401.002,A -85,B 0,C 180,E1 -25553.379,E2 -25553.379} C_VEL
LIN {X 0,Y 177.732,Z 390.368,A -85,B 0,C 180,E1 -25554.781,E2 -25554.781} C_VEL
LIN {X 0,Y 181.564,Z 379.043,A -85,B 0,C 180,E1 -25555.944,E2 -25555.944} C_VEL
LIN {X 0,Y 184.81,Z 366.331,A -85,B 0,C 180,E1 -25556.873,E2 -25556.873} C_VEL
LIN {X 0,Y 187.192,Z 352.056,A -85,B 0,C 180,E1 -25557.519,E2 -25557.519} C_VEL
LIN {X 0,Y 188.793,Z 337.03,A -85,B 0,C 180,E1 -25558.066,E2 -25558.066} C_VEL
LIN {X 0,Y 185.996,Z 330.671,A -85,B 0,C 180,E1 -25561.168,E2 -25561.168} C_VEL
LIN {X 0,Y 183.379,Z 325.364,A -85,B 0,C 180,E1 -25564.848,E2 -25564.848} C_VEL
LIN {X 0,Y 182.727,Z 323.951,A -85,B 0,C 180,E1 -25565.968,E2 -25565.968} C_VEL
LIN {X 0,Y 180.901,Z 321.026,A -85,B 0,C 180,E1 -25570.008,E2 -25570.008} C_VEL
LIN {X 0,Y 180.569,Z 319.974,A -85,B 0,C 180,E1 -25571.234,E2 -25571.234} C_VEL
LIN {X 0,Y 179.93,Z 319.744,A -85,B 0,C 180,E1 -25578.221,E2 -25578.221} C_VEL
LIN {X 0,Y 180.536,Z 320.386,A -85,B 0,C 180,E1 -25581.297,E2 -25581.297} C_VEL
LIN {X 0,Y 182.456,Z 325.271,A -85,B 0,C 180,E1 -25586.382,E2 -25586.382} C_VEL
LIN {X 0,Y 184.288,Z 330.143,A -85,B 0,C 180,E1 -25589.503,E2 -25589.503} C_VEL
LIN {X 0,Y 186.363,Z 335.889,A -85,B 0,C 180,E1 -25592.312,E2 -25592.312} C_VEL
LIN {X 0,Y 188.348,Z 342.182,A -85,B 0,C 180,E1 -25594.669,E2 -25594.669} C_VEL
LIN {X 0,Y 185.674,Z 364.367,A -85,B 0,C 180,E1 -25595.472,E2 -25595.472} C_VEL
LIN {X 0,Y 182.825,Z 377.686,A -85,B 0,C 180,E1 -25596.173,E2 -25596.173} C_VEL
LIN {X 0,Y 179.334,Z 389.116,A -85,B 0,C 180,E1 -25597.017,E2 -25597.017} C_VEL
LIN {X 0,Y 174.575,Z 401.251,A -85,B 0,C 180,E1 -25598.279,E2 -25598.279} C_VEL
LIN {X 0,Y 169.317,Z 412.201,A -85,B 0,C 180,E1 -25599.837,E2 -25599.837} C_VEL
LIN {X 0,Y 163.539,Z 422.216,A -85,B 0,C 180,E1 -25601.698,E2 -25601.698} C_VEL
LIN {X 0,Y 156.83,Z 432.097,A -85,B 0,C 180,E1 -25604.194,E2 -25604.194} C_VEL
LIN {X 0,Y 151.09,Z 439.511,A -85,B 0,C 180,E1 -25606.68,E2 -25606.68} C_VEL
LIN {X 0,Y 144.693,Z 446.85,A -85,B 0,C 180,E1 -25609.943,E2 -25609.943} C_VEL
LIN {X 0,Y 137.956,Z 453.727,A -85,B 0,C 180,E1 -25614.138,E2 -25614.138} C_VEL
LIN {X 0,Y 133.037,Z 458.313,A -85,B 0,C 180,E1 -25618.112,E2 -25618.112} C_VEL
LIN {X 0,Y 128.599,Z 461.863,A -85,B 0,C 180,E1 -25622.321,E2 -25622.321} C_VEL
LIN {X 0,Y 125.01,Z 464.455,A -85,B 0,C 180,E1 -25626.826,E2 -25626.826} C_VEL
LIN {X 0,Y 123.031,Z 465.711,A -85,B 0,C 180,E1 -25629.957,E2 -25629.957} C_VEL
LIN {X 0,Y 120.494,Z 467.021,A -85,B 0,C 180,E1 -25636.509,E2 -25636.509} C_VEL
LIN {X 0,Y 119.43,Z 466.834,A -85,B 0,C 180,E1 -25643.241,E2 -25643.241} C_VEL
LIN {X 0,Y 119.383,Z 466.169,A -85,B 0,C 180,E1 -25646.625,E2 -25646.625} C_VEL
LIN {X 0,Y 119.511,Z 464.905,A -85,B 0,C 180,E1 -25650.379,E2 -25650.379} C_VEL
LIN {X 0,Y 119.453,Z 463.509,A -85,B 0,C 180,E1 -25653.373,E2 -25653.373} C_VEL
LIN {X 0,Y 119.678,Z 460.318,A -85,B 0,C 180,E1 -25658.442,E2 -25658.442} C_VEL
LIN {X 0,Y 120.489,Z 456.003,A -85,B 0,C 180,E1 -25663.492,E2 -25663.492} C_VEL
LIN {X 0,Y 121.441,Z 452.481,A -85,B 0,C 180,E1 -25666.811,E2 -25666.811} C_VEL
LIN {X 0,Y 121.702,Z 449.593,A -85,B 0,C 180,E1 -25669.243,E2 -25669.243} C_VEL
LIN {X 0,Y 120.717,Z 444.245,A -85,B 0,C 180,E1 -25673.177,E2 -25673.177} C_VEL
LIN {X 0,Y 120.174,Z 438.222,A -85,B 0,C 180,E1 -25676.939,E2 -25676.939} C_VEL
LIN {X 0,Y 121.1,Z 434.275,A -85,B 0,C 180,E1 -25678.994,E2 -25678.994} C_VEL
LIN {X 0,Y 124.281,Z 426.063,A -85,B 0,C 180,E1 -25682.494,E2 -25682.494} C_VEL
LIN {X 0,Y 127.751,Z 416.292,A -85,B 0,C 180,E1 -25685.768,E2 -25685.768} C_VEL
LIN {X 0,Y 131.306,Z 405.677,A -85,B 0,C 180,E1 -25688.477,E2 -25688.477} C_VEL
LIN {X 0,Y 134.582,Z 393.84,A -85,B 0,C 180,E1 -25690.749,E2 -25690.749} C_VEL
LIN {X 0,Y 137.358,Z 381.716,A -85,B 0,C 180,E1 -25692.433,E2 -25692.433} C_VEL
LIN {X 0,Y 139.544,Z 368.632,A -85,B 0,C 180,E1 -25693.703,E2 -25693.703} C_VEL
LIN {X 0,Y 141.019,Z 353.745,A -85,B 0,C 180,E1 -25694.566,E2 -25694.566} C_VEL
LIN {X 0,Y 143.243,Z 322.336,A -85,B 0,C 180,E1 -25696.112,E2 -25696.112} C_VEL
LIN {X 0,Y 142.72,Z 316.743,A -85,B 0,C 180,E1 -25696.653,E2 -25696.653} C_VEL
LIN {X 0,Y 137.508,Z 301.602,A -85,B 0,C 180,E1 -25699.389,E2 -25699.389} C_VEL
LIN {X 0,Y 132.519,Z 289.447,A -85,B 0,C 180,E1 -25702.116,E2 -25702.116} C_VEL
LIN {X 0,Y 129.219,Z 282.62,A -85,B 0,C 180,E1 -25703.967,E2 -25703.967} C_VEL
LIN {X 0,Y 123.571,Z 273.493,A -85,B 0,C 180,E1 -25707.276,E2 -25707.276} C_VEL
LIN {X 0,Y 120.785,Z 269.456,A -85,B 0,C 180,E1 -25709.027,E2 -25709.027} C_VEL
LIN {X 0,Y 118.534,Z 266.235,A -85,B 0,C 180,E1 -25710.534,E2 -25710.534} C_VEL
LIN {X 0,Y 117.917,Z 265.194,A -85,B 0,C 180,E1 -25710.979,E2 -25710.979} C_VEL
LIN {X 0,Y 115.813,Z 262.982,A -85,B 0,C 180,E1 -25712.417,E2 -25712.417} C_VEL
LIN {X 0,Y 114.801,Z 260.176,A -85,B 0,C 180,E1 -25713.386,E2 -25713.386} C_VEL
LIN {X 0,Y 114.942,Z 260.147,A -85,B 0,C 180,E1 -25718.458,E2 -25718.458} C_VEL
LIN {X 0,Y 115.085,Z 260.128,A -85,B 0,C 180,E1 -25725.842,E2 -25725.842} C_VEL
LIN {X 0,Y 115.307,Z 260.121,A -85,B 0,C 180,E1 -25729.445,E2 -25729.445} C_VEL
LIN {X 0,Y 115.451,Z 260.033,A -85,B 0,C 180,E1 -25736.49,E2 -25736.49} C_VEL
LIN {X 0,Y 115.929,Z 259.998,A -85,B 0,C 180,E1 -25739.98,E2 -25739.98} C_VEL
LIN {X 0,Y 115.338,Z 260.11,A -85,B 0,C 180,E1 -25746.98,E2 -25746.98} C_VEL
LIN {X 0,Y 115.195,Z 260.132,A -85,B 0,C 180,E1 -25752.543,E2 -25752.543} C_VEL
LIN {X 0,Y 114.976,Z 260.143,A -85,B 0,C 180,E1 -25757.774,E2 -25757.774} C_VEL
LIN {X 0,Y 114.925,Z 260.167,A -85,B 0,C 180,E1 -25763.47,E2 -25763.47} C_VEL
LIN {X 0,Y 114.829,Z 260.108,A -85,B 0,C 180,E1 -25771.037,E2 -25771.037} C_VEL
LIN {X 0,Y 114.745,Z 260.183,A -85,B 0,C 180,E1 -25777.742,E2 -25777.742} C_VEL
LIN {X 0,Y 114.735,Z 260.18,A -85,B 0,C 180,E1 -25782.69,E2 -25782.69} C_VEL
LIN {X 0,Y 114.751,Z 260.191,A -85,B 0,C 180,E1 -25787.648,E2 -25787.648} C_VEL
LIN {X 0,Y 114.747,Z 260.191,A -85,B 0,C 180,E1 -25792.733,E2 -25792.733} C_VEL
LIN {X 0,Y 114.859,Z 260.184,A -85,B 0,C 180,E1 -25799.823,E2 -25799.823} C_VEL
LIN {X 0,Y 114.842,Z 260.241,A -85,B 0,C 180,E1 -25800.362,E2 -25800.362} C_VEL
LIN {X 0,Y 115.698,Z 262.826,A -85,B 0,C 180,E1 -25801.17,E2 -25801.17} C_VEL
LIN {X 0,Y 117.719,Z 265.021,A -85,B 0,C 180,E1 -25802.571,E2 -25802.571} C_VEL
LIN {X 0,Y 118.419,Z 265.912,A -85,B 0,C 180,E1 -25803.05,E2 -25803.05} C_VEL
LIN {X 0,Y 120.611,Z 269.229,A -85,B 0,C 180,E1 -25804.539,E2 -25804.539} C_VEL
LIN {X 0,Y 122.003,Z 271.041,A -85,B 0,C 180,E1 -25805.408,E2 -25805.408} C_VEL
LIN {X 0,Y 124.981,Z 275.462,A -85,B 0,C 180,E1 -25807.234,E2 -25807.234} C_VEL
LIN {X 0,Y 131.264,Z 285.555,A -85,B 0,C 180,E1 -25810.767,E2 -25810.767} C_VEL
LIN {X 0,Y 136.108,Z 294.175,A -85,B 0,C 180,E1 -25813.223,E2 -25813.223} C_VEL
LIN {X 0,Y 143.662,Z 309.904,A -85,B 0,C 180,E1 -25816.819,E2 -25816.819} C_VEL
LIN {X 0,Y 144.069,Z 311.113,A -85,B 0,C 180,E1 -25817.023,E2 -25817.023} C_VEL
LIN {X 0,Y 140.366,Z 356.144,A -85,B 0,C 180,E1 -25819.204,E2 -25819.204} C_VEL
LIN {X 0,Y 138.485,Z 369.16,A -85,B 0,C 180,E1 -25820.319,E2 -25820.319} C_VEL
LIN {X 0,Y 136.423,Z 380.339,A -85,B 0,C 180,E1 -25821.757,E2 -25821.757} C_VEL
LIN {X 0,Y 133.32,Z 392.948,A -85,B 0,C 180,E1 -25823.948,E2 -25823.948} C_VEL
LIN {X 0,Y 130.061,Z 403.941,A -85,B 0,C 180,E1 -25826.515,E2 -25826.515} C_VEL
LIN {X 0,Y 126.458,Z 414.517,A -85,B 0,C 180,E1 -25829.723,E2 -25829.723} C_VEL
LIN {X 0,Y 122.971,Z 423.602,A -85,B 0,C 180,E1 -25833.276,E2 -25833.276} C_VEL
LIN {X 0,Y 119.758,Z 431.93,A -85,B 0,C 180,E1 -25837.502,E2 -25837.502} C_VEL
LIN {X 0,Y 116.945,Z 439.089,A -85,B 0,C 180,E1 -25842.142,E2 -25842.142} C_VEL
LIN {X 0,Y 114.558,Z 445.857,A -85,B 0,C 180,E1 -25847.862,E2 -25847.862} C_VEL
LIN {X 0,Y 112.972,Z 451.101,A -85,B 0,C 180,E1 -25853.85,E2 -25853.85} C_VEL
LIN {X 0,Y 111.959,Z 455.043,A -85,B 0,C 180,E1 -25860.143,E2 -25860.143} C_VEL
LIN {X 0,Y 111.887,Z 457.26,A -85,B 0,C 180,E1 -25865.297,E2 -25865.297} C_VEL
LIN {X 0,Y 112.856,Z 458.847,A -85,B 0,C 180,E1 -25871.678,E2 -25871.678} C_VEL
LIN {X 0,Y 114.812,Z 459.215,A -85,B 0,C 180,E1 -25877.704,E2 -25877.704} C_VEL
LIN {X 0,Y 117.75,Z 458.473,A -85,B 0,C 180,E1 -25883.382,E2 -25883.382} C_VEL
LIN {X 0,Y 122.3,Z 456.278,A -85,B 0,C 180,E1 -25889.537,E2 -25889.537} C_VEL
LIN {X 0,Y 127.968,Z 452.604,A -85,B 0,C 180,E1 -25895.079,E2 -25895.079} C_VEL
LIN {X 0,Y 134.619,Z 447.491,A -85,B 0,C 180,E1 -25899.999,E2 -25899.999} C_VEL
LIN {X 0,Y 140.891,Z 441.818,A -85,B 0,C 180,E1 -25903.783,E2 -25903.783} C_VEL
LIN {X 0,Y 147.727,Z 434.657,A -85,B 0,C 180,E1 -25907.218,E2 -25907.218} C_VEL
LIN {X 0,Y 154.334,Z 426.618,A -85,B 0,C 180,E1 -25910.081,E2 -25910.081} C_VEL
LIN {X 0,Y 161.305,Z 416.755,A -85,B 0,C 180,E1 -25912.672,E2 -25912.672} C_VEL
LIN {X 0,Y 167.604,Z 405.98,A -85,B 0,C 180,E1 -25914.785,E2 -25914.785} C_VEL
LIN {X 0,Y 173.381,Z 393.995,A -85,B 0,C 180,E1 -25916.509,E2 -25916.509} C_VEL
LIN {X 0,Y 178.133,Z 381.257,A -85,B 0,C 180,E1 -25917.845,E2 -25917.845} C_VEL
LIN {X 0,Y 181.868,Z 367.719,A -85,B 0,C 180,E1 -25918.858,E2 -25918.858} C_VEL
LIN {X 0,Y 184.183,Z 355.145,A -85,B 0,C 180,E1 -25919.453,E2 -25919.453} C_VEL
LIN {X 0,Y 185.834,Z 341.009,A -85,B 0,C 180,E1 -25919.943,E2 -25919.943} C_VEL
LIN {X 0,Y 183.934,Z 336.514,A -85,B 0,C 180,E1 -25922.339,E2 -25922.339} C_VEL
LIN {X 0,Y 181.732,Z 331.656,A -85,B 0,C 180,E1 -25925.785,E2 -25925.785} C_VEL
LIN {X 0,Y 181.071,Z 330.397,A -85,B 0,C 180,E1 -25927.064,E2 -25927.064} C_VEL
LIN {X 0,Y 179.606,Z 327.478,A -85,B 0,C 180,E1 -25930.898,E2 -25930.898} C_VEL
LIN {X 0,Y 179.427,Z 326.955,A -85,B 0,C 180,E1 -25931.706,E2 -25931.706} C_VEL
LIN {X 0,Y 178.935,Z 326.786,A -85,B 0,C 180,E1 -25938.326,E2 -25938.326} C_VEL
LIN {X 0,Y 179.403,Z 327.33,A -85,B 0,C 180,E1 -25940.906,E2 -25940.906} C_VEL
LIN {X 0,Y 180.976,Z 331.776,A -85,B 0,C 180,E1 -25945.593,E2 -25945.593} C_VEL
LIN {X 0,Y 182.573,Z 336.474,A -85,B 0,C 180,E1 -25948.622,E2 -25948.622} C_VEL
LIN {X 0,Y 184.219,Z 341.588,A -85,B 0,C 180,E1 -25951.17,E2 -25951.17} C_VEL
LIN {X 0,Y 185.426,Z 345.607,A -85,B 0,C 180,E1 -25952.766,E2 -25952.766} C_VEL
LIN {X 0,Y 182.961,Z 364.645,A -85,B 0,C 180,E1 -25953.438,E2 -25953.438} C_VEL
LIN {X 0,Y 180.379,Z 376.395,A -85,B 0,C 180,E1 -25954.041,E2 -25954.041} C_VEL
LIN {X 0,Y 176.675,Z 388.377,A -85,B 0,C 180,E1 -25954.873,E2 -25954.873} C_VEL
LIN {X 0,Y 171.748,Z 400.566,A -85,B 0,C 180,E1 -25956.084,E2 -25956.084} C_VEL
LIN {X 0,Y 166.275,Z 411.551,A -85,B 0,C 180,E1 -25957.581,E2 -25957.581} C_VEL
LIN {X 0,Y 160.252,Z 421.614,A -85,B 0,C 180,E1 -25959.382,E2 -25959.382} C_VEL
LIN {X 0,Y 153.279,Z 431.56,A -85,B 0,C 180,E1 -25961.836,E2 -25961.836} C_VEL
LIN {X 0,Y 147.187,Z 439.032,A -85,B 0,C 180,E1 -25964.258,E2 -25964.258} C_VEL
LIN {X 0,Y 140.451,Z 446.398,A -85,B 0,C 180,E1 -25967.507,E2 -25967.507} C_VEL
LIN {X 0,Y 134.2,Z 452.382,A -85,B 0,C 180,E1 -25971.067,E2 -25971.067} C_VEL
LIN {X 0,Y 128.74,Z 457.144,A -85,B 0,C 180,E1 -25974.997,E2 -25974.997} C_VEL
LIN {X 0,Y 123.832,Z 460.923,A -85,B 0,C 180,E1 -25979.285,E2 -25979.285} C_VEL
LIN {X 0,Y 118.503,Z 464.468,A -85,B 0,C 180,E1 -25985.472,E2 -25985.472} C_VEL
LIN {X 0,Y 114.753,Z 466.383,A -85,B 0,C 180,E1 -25992.169,E2 -25992.169} C_VEL
LIN {X 0,Y 112.777,Z 466.819,A -85,B 0,C 180,E1 -25999.225,E2 -25999.225} C_VEL
LIN {X 0,Y 112.36,Z 466.474,A -85,B 0,C 180,E1 -26002.814,E2 -26002.814} C_VEL
LIN {X 0,Y 112.291,Z 465.707,A -85,B 0,C 180,E1 -26006.412,E2 -26006.412} C_VEL
LIN {X 0,Y 112.481,Z 464.543,A -85,B 0,C 180,E1 -26010,E2 -26010} C_VEL
LIN {X 0,Y 112.394,Z 461.932,A -85,B 0,C 180,E1 -26015.382,E2 -26015.382} C_VEL
LIN {X 0,Y 112.866,Z 458.249,A -85,B 0,C 180,E1 -26020.766,E2 -26020.766} C_VEL
LIN {X 0,Y 114.042,Z 453.39,A -85,B 0,C 180,E1 -26026.1,E2 -26026.1} C_VEL
LIN {X 0,Y 116.174,Z 447.234,A -85,B 0,C 180,E1 -26031.282,E2 -26031.282} C_VEL
LIN {X 0,Y 119.12,Z 439.541,A -85,B 0,C 180,E1 -26036.263,E2 -26036.263} C_VEL
LIN {X 0,Y 121.1,Z 434.275,A -85,B 0,C 180,E1 -26038.994,E2 -26038.994} C_VEL
LIN {X 0,Y 122.069,Z 430.207,A -85,B 0,C 180,E1 -26040.938,E2 -26040.938} C_VEL
LIN {X 0,Y 121.99,Z 423.137,A -85,B 0,C 180,E1 -26044.201,E2 -26044.201} C_VEL
LIN {X 0,Y 122.088,Z 415.561,A -85,B 0,C 180,E1 -26047.239,E2 -26047.239} C_VEL
LIN {X 0,Y 123.287,Z 410.655,A -85,B 0,C 180,E1 -26048.739,E2 -26048.739} C_VEL
LIN {X 0,Y 126.755,Z 400.003,A -85,B 0,C 180,E1 -26051.178,E2 -26051.178} C_VEL
LIN {X 0,Y 130.102,Z 387.58,A -85,B 0,C 180,E1 -26053.263,E2 -26053.263} C_VEL
LIN {X 0,Y 132.698,Z 374.619,A -85,B 0,C 180,E1 -26054.833,E2 -26054.833} C_VEL
LIN {X 0,Y 134.511,Z 362.167,A -85,B 0,C 180,E1 -26055.788,E2 -26055.788} C_VEL
LIN {X 0,Y 137.524,Z 323.556,A -85,B 0,C 180,E1 -26057.75,E2 -26057.75} C_VEL
LIN {X 0,Y 137.003,Z 318.696,A -85,B 0,C 180,E1 -26058.277,E2 -26058.277} C_VEL
LIN {X 0,Y 132.424,Z 304.968,A -85,B 0,C 180,E1 -26060.913,E2 -26060.913} C_VEL
LIN {X 0,Y 127.422,Z 292.705,A -85,B 0,C 180,E1 -26063.84,E2 -26063.84} C_VEL
LIN {X 0,Y 124.84,Z 287.127,A -85,B 0,C 180,E1 -26065.437,E2 -26065.437} C_VEL
LIN {X 0,Y 119.067,Z 277.805,A -85,B 0,C 180,E1 -26069.084,E2 -26069.084} C_VEL
LIN {X 0,Y 116.934,Z 274.653,A -85,B 0,C 180,E1 -26070.534,E2 -26070.534} C_VEL
LIN {X 0,Y 114.112,Z 270.614,A -85,B 0,C 180,E1 -26072.593,E2 -26072.593} C_VEL
LIN {X 0,Y 111.825,Z 267.452,A -85,B 0,C 180,E1 -26074.396,E2 -26074.396} C_VEL
LIN {X 0,Y 111.172,Z 266.252,A -85,B 0,C 180,E1 -26074.959,E2 -26074.959} C_VEL
LIN {X 0,Y 109.084,Z 264.229,A -85,B 0,C 180,E1 -26076.627,E2 -26076.627} C_VEL
LIN {X 0,Y 107.986,Z 261.659,A -85,B 0,C 180,E1 -26077.751,E2 -26077.751} C_VEL
LIN {X 0,Y 107.885,Z 261.03,A -85,B 0,C 180,E1 -26077.981,E2 -26077.981} C_VEL
LIN {X 0,Y 107.974,Z 260.999,A -85,B 0,C 180,E1 -26084.888,E2 -26084.888} C_VEL
LIN {X 0,Y 108.227,Z 261.004,A -85,B 0,C 180,E1 -26088.745,E2 -26088.745} C_VEL
LIN {X 0,Y 108.28,Z 260.958,A -85,B 0,C 180,E1 -26092.521,E2 -26092.521} C_VEL
LIN {X 0,Y 108.858,Z 260.875,A -85,B 0,C 180,E1 -26099.979,E2 -26099.979} C_VEL
LIN {X 0,Y 108.278,Z 260.986,A -85,B 0,C 180,E1 -26107.437,E2 -26107.437} C_VEL
LIN {X 0,Y 108.128,Z 261.013,A -85,B 0,C 180,E1 -26112.855,E2 -26112.855} C_VEL
LIN {X 0,Y 107.874,Z 261.026,A -85,B 0,C 180,E1 -26118.988,E2 -26118.988} C_VEL
LIN {X 0,Y 107.834,Z 261.048,A -85,B 0,C 180,E1 -26124.158,E2 -26124.158} C_VEL
LIN {X 0,Y 107.752,Z 260.988,A -85,B 0,C 180,E1 -26132.017,E2 -26132.017} C_VEL
LIN {X 0,Y 107.652,Z 261.071,A -85,B 0,C 180,E1 -26138.427,E2 -26138.427} C_VEL
LIN {X 0,Y 107.633,Z 261.074,A -85,B 0,C 180,E1 -26145.877,E2 -26145.877} C_VEL
LIN {X 0,Y 107.646,Z 261.066,A -85,B 0,C 180,E1 -26151.54,E2 -26151.54} C_VEL
LIN {X 0,Y 107.698,Z 261.184,A -85,B 0,C 180,E1 -26155.634,E2 -26155.634} C_VEL
LIN {X 0,Y 108.634,Z 263.745,A -85,B 0,C 180,E1 -26156.655,E2 -26156.655} C_VEL
LIN {X 0,Y 110.624,Z 265.914,A -85,B 0,C 180,E1 -26158.302,E2 -26158.302} C_VEL
LIN {X 0,Y 111.529,Z 266.78,A -85,B 0,C 180,E1 -26159.004,E2 -26159.004} C_VEL
LIN {X 0,Y 113.557,Z 270.025,A -85,B 0,C 180,E1 -26160.672,E2 -26160.672} C_VEL
LIN {X 0,Y 115.031,Z 271.765,A -85,B 0,C 180,E1 -26161.755,E2 -26161.755} C_VEL
LIN {X 0,Y 117.638,Z 275.388,A -85,B 0,C 180,E1 -26163.605,E2 -26163.605} C_VEL
LIN {X 0,Y 122.814,Z 283.361,A -85,B 0,C 180,E1 -26166.953,E2 -26166.953} C_VEL
LIN {X 0,Y 129.912,Z 295.467,A -85,B 0,C 180,E1 -26171.06,E2 -26171.06} C_VEL
LIN {X 0,Y 138.197,Z 312.795,A -85,B 0,C 180,E1 -26175.338,E2 -26175.338} C_VEL
LIN {X 0,Y 134.521,Z 356.402,A -85,B 0,C 180,E1 -26177.524,E2 -26177.524} C_VEL
LIN {X 0,Y 132.621,Z 369.114,A -85,B 0,C 180,E1 -26178.635,E2 -26178.635} C_VEL
LIN {X 0,Y 130.2,Z 381.568,A -85,B 0,C 180,E1 -26180.289,E2 -26180.289} C_VEL
LIN {X 0,Y 127.242,Z 392.97,A -85,B 0,C 180,E1 -26182.351,E2 -26182.351} C_VEL
LIN {X 0,Y 123.677,Z 404.41,A -85,B 0,C 180,E1 -26185.11,E2 -26185.11} C_VEL
LIN {X 0,Y 119.748,Z 415.423,A -85,B 0,C 180,E1 -26188.623,E2 -26188.623} C_VEL
LIN {X 0,Y 115.907,Z 424.897,A -85,B 0,C 180,E1 -26192.606,E2 -26192.606} C_VEL
LIN {X 0,Y 112.502,Z 433.226,A -85,B 0,C 180,E1 -26197.177,E2 -26197.177} C_VEL
LIN {X 0,Y 109.412,Z 440.833,A -85,B 0,C 180,E1 -26202.616,E2 -26202.616} C_VEL
LIN {X 0,Y 107.608,Z 445.677,A -85,B 0,C 180,E1 -26207.091,E2 -26207.091} C_VEL
LIN {X 0,Y 105.91,Z 451.049,A -85,B 0,C 180,E1 -26213.462,E2 -26213.462} C_VEL
LIN {X 0,Y 104.909,Z 454.742,A -85,B 0,C 180,E1 -26219.489,E2 -26219.489} C_VEL
LIN {X 0,Y 104.873,Z 457.63,A -85,B 0,C 180,E1 -26226.511,E2 -26226.511} C_VEL
LIN {X 0,Y 106.097,Z 459.163,A -85,B 0,C 180,E1 -26233.261,E2 -26233.261} C_VEL
LIN {X 0,Y 108.923,Z 459.446,A -85,B 0,C 180,E1 -26240.737,E2 -26240.737} C_VEL
LIN {X 0,Y 111.688,Z 458.713,A -85,B 0,C 180,E1 -26245.533,E2 -26245.533} C_VEL
LIN {X 0,Y 115.938,Z 456.887,A -85,B 0,C 180,E1 -26251.015,E2 -26251.015} C_VEL
LIN {X 0,Y 122.197,Z 453.289,A -85,B 0,C 180,E1 -26256.953,E2 -26256.953} C_VEL
LIN {X 0,Y 129.316,Z 448.24,A -85,B 0,C 180,E1 -26262.033,E2 -26262.033} C_VEL
LIN {X 0,Y 135.406,Z 443.157,A -85,B 0,C 180,E1 -26265.568,E2 -26265.568} C_VEL
LIN {X 0,Y 143.057,Z 435.779,A -85,B 0,C 180,E1 -26269.27,E2 -26269.27} C_VEL
LIN {X 0,Y 150.51,Z 427.259,A -85,B 0,C 180,E1 -26272.33,E2 -26272.33} C_VEL
LIN {X 0,Y 157.926,Z 417.316,A -85,B 0,C 180,E1 -26274.909,E2 -26274.909} C_VEL
LIN {X 0,Y 164.177,Z 407.129,A -85,B 0,C 180,E1 -26276.889,E2 -26276.889} C_VEL
LIN {X 0,Y 169.61,Z 396.502,A -85,B 0,C 180,E1 -26278.418,E2 -26278.418} C_VEL
LIN {X 0,Y 174.73,Z 383.989,A -85,B 0,C 180,E1 -26279.765,E2 -26279.765} C_VEL
LIN {X 0,Y 178.658,Z 370.922,A -85,B 0,C 180,E1 -26280.787,E2 -26280.787} C_VEL
LIN {X 0,Y 181.457,Z 357.739,A -85,B 0,C 180,E1 -26281.449,E2 -26281.449} C_VEL
LIN {X 0,Y 183.061,Z 345.04,A -85,B 0,C 180,E1 -26281.928,E2 -26281.928} C_VEL
LIN {X 0,Y 181.637,Z 341.572,A -85,B 0,C 180,E1 -26284.061,E2 -26284.061} C_VEL
LIN {X 0,Y 180.057,Z 337.58,A -85,B 0,C 180,E1 -26287.012,E2 -26287.012} C_VEL
LIN {X 0,Y 178.462,Z 334.343,A -85,B 0,C 180,E1 -26291.368,E2 -26291.368} C_VEL
LIN {X 0,Y 178.283,Z 333.906,A -85,B 0,C 180,E1 -26292.259,E2 -26292.259} C_VEL
LIN {X 0,Y 177.941,Z 333.834,A -85,B 0,C 180,E1 -26298.432,E2 -26298.432} C_VEL
LIN {X 0,Y 178.306,Z 334.312,A -85,B 0,C 180,E1 -26300.56,E2 -26300.56} C_VEL
LIN {X 0,Y 179.609,Z 338.426,A -85,B 0,C 180,E1 -26304.909,E2 -26304.909} C_VEL
LIN {X 0,Y 180.985,Z 343.077,A -85,B 0,C 180,E1 -26307.883,E2 -26307.883} C_VEL
LIN {X 0,Y 182.289,Z 347.613,A -85,B 0,C 180,E1 -26310.144,E2 -26310.144} C_VEL
LIN {X 0,Y 182.673,Z 349.143,A -85,B 0,C 180,E1 -26310.781,E2 -26310.781} C_VEL
LIN {X 0,Y 180.43,Z 365.268,A -85,B 0,C 180,E1 -26311.365,E2 -26311.365} C_VEL
LIN {X 0,Y 177.789,Z 376.63,A -85,B 0,C 180,E1 -26311.924,E2 -26311.924} C_VEL
